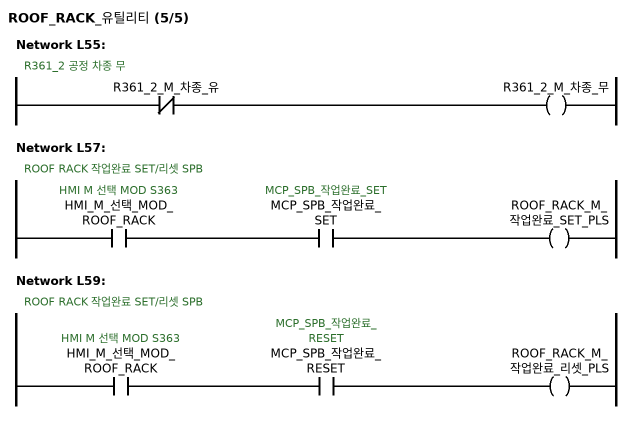
(* [picture p72: ROOF_RACK_유틸리티 rungs L55-L59] *)
(* R361_2 공정 차종 무 *)
(* Rung L55 *)
R361_2_M_차종_무 := NOT R361_2_M_차종_유;
(* ROOF RACK 작업완료 SET/리셋 SPB *)
(* Rung L57 *)
ROOF_RACK_M_작업완료_SET_PLS := HMI_M_선택_MOD_ROOF_RACK AND MCP_SPB_작업완료_SET;
(* ROOF RACK 작업완료 SET/리셋 SPB *)
(* Rung L59 *)
ROOF_RACK_M_작업완료_리셋_PLS := HMI_M_선택_MOD_ROOF_RACK AND MCP_SPB_작업완료_RESET;
END_PROGRAM

PROGRAM ROOF_RACK_차종입력_차종삭제 (* task: 스캔 프로그램 *)
VAR
    INST : TON;
    INST1 : TON;
    INST2 : TON;
    INST3 : TON;
    INST4 : TON;
    INST5 : TON;
END_VAR
VAR_EXTERNAL
    R361_1_I_RB_PLT_최종UNLOAD_완료 : BOOL; (* AT %MW84013.12 *) (* R361_1_I_RB_PLT_최종UNLOAD_완료 *)
    R361_2_I_RB_PLT_최종UNLOAD_완료 : BOOL; (* AT %MW84023.12 *) (* R361_2_I_RB_PLT_최종UNLOAD_완료 *)
END_VAR
VAR_EXTERNAL RETAIN
    R361_1_M_RACK3_프로그램_OK : BOOL; (* AT %MW1563.2 *)
    R361_1_M_RACK4_프로그램_OK : BOOL; (* AT %MW1563.3 *)
    R361_1_M_RACK5_프로그램_OK : BOOL; (* AT %MW1563.4 *)
    R361_1_M_RACK6_프로그램_OK : BOOL; (* AT %MW1563.5 *)
    R361_2_M_RACK1_프로그램_OK : BOOL; (* AT %MW1563.0 *)
    R361_2_M_RACK2_프로그램_OK : BOOL; (* AT %MW1563.1 *)
    ROOF_RACK1_M_HMI입력_차종 : WORD; (* AT %MW501 *)
    ROOF_RACK1_M_랙감지_유 : BOOL; (* AT %MW1501.0 *)
    ROOF_RACK1_M_로딩완료 : BOOL; (* AT %MW1561.0 *)
    ROOF_RACK1_M_막장감지_유 : BOOL; (* AT %MW1503.0 *)
    ROOF_RACK1_M_제품수량 : WORD; (* AT %MW511 *)
    ROOF_RACK1_M_차종 : WORD; (* AT %MW1541 *)
    ROOF_RACK2_M_HMI입력_차종 : WORD; (* AT %MW502 *)
    ROOF_RACK2_M_랙감지_유 : BOOL; (* AT %MW1501.2 *)
    ROOF_RACK2_M_로딩완료 : BOOL; (* AT %MW1561.1 *)
    ROOF_RACK2_M_막장감지_유 : BOOL; (* AT %MW1503.2 *)
    ROOF_RACK2_M_제품수량 : WORD; (* AT %MW512 *)
    ROOF_RACK2_M_차종 : WORD; (* AT %MW1542 *)
    ROOF_RACK3_M_HMI입력_차종 : WORD; (* AT %MW503 *)
    ROOF_RACK3_M_랙감지_유 : BOOL; (* AT %MW1501.4 *)
    ROOF_RACK3_M_로딩완료 : BOOL; (* AT %MW1561.2 *)
    ROOF_RACK3_M_막장감지_유 : BOOL; (* AT %MW1503.4 *)
    ROOF_RACK3_M_제품수량 : WORD; (* AT %MW513 *)
    ROOF_RACK3_M_차종 : WORD; (* AT %MW1543 *)
    ROOF_RACK4_M_HMI입력_차종 : WORD; (* AT %MW504 *)
    ROOF_RACK4_M_랙감지_유 : BOOL; (* AT %MW1501.6 *)
    ROOF_RACK4_M_로딩완료 : BOOL; (* AT %MW1561.3 *)
    ROOF_RACK4_M_막장감지_유 : BOOL; (* AT %MW1503.6 *)
    ROOF_RACK4_M_제품수량 : WORD; (* AT %MW514 *)
    ROOF_RACK4_M_차종 : WORD; (* AT %MW1544 *)
    ROOF_RACK5_M_HMI입력_차종 : WORD; (* AT %MW505 *)
    ROOF_RACK5_M_랙감지_유 : BOOL; (* AT %MW1501.8 *)
    ROOF_RACK5_M_로딩완료 : BOOL; (* AT %MW1561.4 *)
    ROOF_RACK5_M_막장감지_유 : BOOL; (* AT %MW1503.8 *)
    ROOF_RACK5_M_제품수량 : WORD; (* AT %MW515 *)
    ROOF_RACK5_M_차종 : WORD; (* AT %MW1545 *)
    ROOF_RACK6_M_HMI입력_차종 : WORD; (* AT %MW506 *)
    ROOF_RACK6_M_랙감지_유 : BOOL; (* AT %MW1501.10 *)
    ROOF_RACK6_M_로딩완료 : BOOL; (* AT %MW1561.5 *)
    ROOF_RACK6_M_막장감지_유 : BOOL; (* AT %MW1503.10 *)
    ROOF_RACK6_M_제품수량 : WORD; (* AT %MW516 *)
    ROOF_RACK6_M_차종 : WORD; (* AT %MW1546 *)
END_VAR
VAR
    _p1 : BOOL;
    _p2 : BOOL;
    _p3 : BOOL;
    _p4 : BOOL;
    _p5 : BOOL;
    _p6 : BOOL;
END_VAR
(* ================================================================= *)
(* ROOF RACK 차종 입력 *)
(* ================================================================= *)
(* ROOF RACK1 차종입력 *)
(* Rung L4: network not rendered *)
(* not connected or not rendered: ROOF_RACK1_M_로딩완료, ROOF_RACK1_M_랙감지_유, ROOF_RACK1_M_막장감지_유, ROOF_RACK1_M_HMI입력_차종, ROOF_RACK1_M_차종, 10, ROOF_RACK1_M_제품수량 *)
(* ROOF RACK2 차종입력 *)
(* Rung L8: network not rendered *)
(* not connected or not rendered: ROOF_RACK2_M_로딩완료, ROOF_RACK2_M_랙감지_유, ROOF_RACK2_M_막장감지_유, ROOF_RACK2_M_HMI입력_차종, ROOF_RACK2_M_차종, 10, ROOF_RACK2_M_제품수량 *)
(* ROOF RACK3 차종입력 *)
(* Rung L12: network not rendered *)
(* not connected or not rendered: ROOF_RACK3_M_로딩완료, ROOF_RACK3_M_랙감지_유, ROOF_RACK3_M_막장감지_유, ROOF_RACK3_M_HMI입력_차종, ROOF_RACK3_M_차종, 10, ROOF_RACK3_M_제품수량 *)
(* ROOF RACK4 차종입력 *)
(* Rung L16: network not rendered *)
(* not connected or not rendered: ROOF_RACK4_M_로딩완료, ROOF_RACK4_M_랙감지_유, ROOF_RACK4_M_막장감지_유, ROOF_RACK4_M_HMI입력_차종, ROOF_RACK4_M_차종, 10, ROOF_RACK4_M_제품수량 *)
(* ROOF RACK5 차종입력 *)
(* Rung L20: network not rendered *)
(* not connected or not rendered: ROOF_RACK5_M_로딩완료, ROOF_RACK5_M_랙감지_유, ROOF_RACK5_M_막장감지_유, ROOF_RACK5_M_HMI입력_차종, ROOF_RACK5_M_차종, 10, ROOF_RACK5_M_제품수량 *)
(* ROOF RACK6 차종입력 *)
(* Rung L24: network not rendered *)
(* not connected or not rendered: ROOF_RACK6_M_로딩완료, ROOF_RACK6_M_랙감지_유, ROOF_RACK6_M_막장감지_유, ROOF_RACK6_M_HMI입력_차종, ROOF_RACK6_M_차종, 10, ROOF_RACK6_M_제품수량 *)

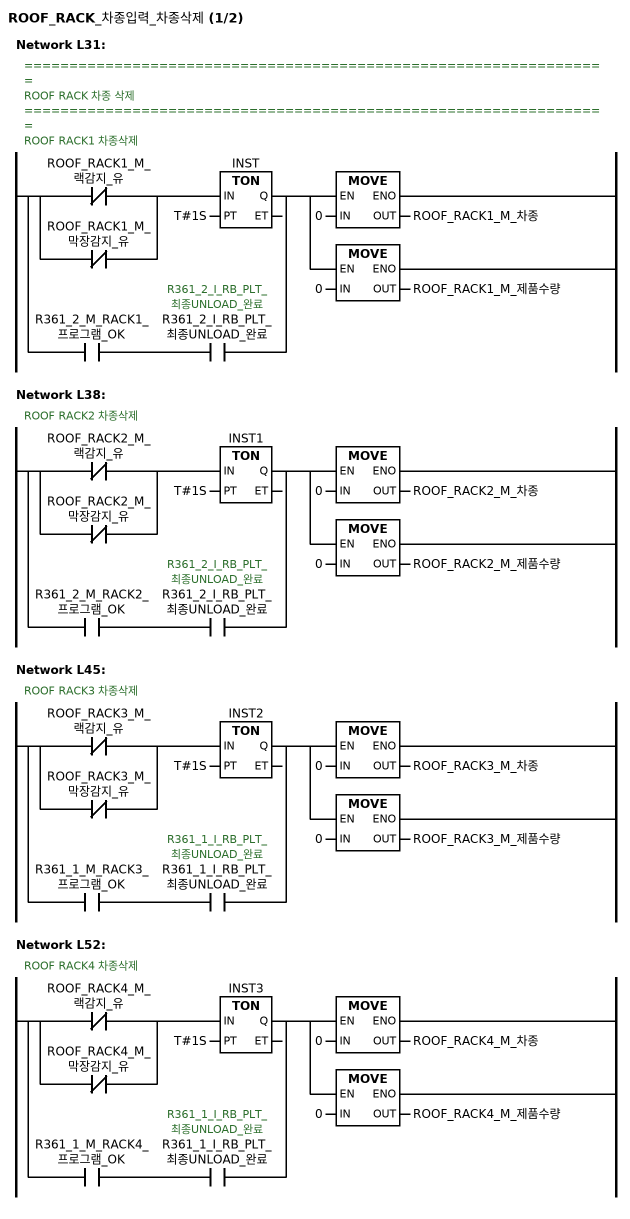
(* ================================================================= *)
(* ROOF RACK 차종 삭제 *)
(* ================================================================= *)
(* ROOF RACK1 차종삭제 *)
(* Rung L31 *)
INST(IN := NOT ROOF_RACK1_M_랙감지_유 OR NOT ROOF_RACK1_M_막장감지_유, PT := T#1S);
_p1 := INST.Q OR (R361_2_M_RACK1_프로그램_OK AND R361_2_I_RB_PLT_최종UNLOAD_완료);
IF _p1 THEN
    ROOF_RACK1_M_차종 := 0;
    ROOF_RACK1_M_제품수량 := 0;
END_IF;
(* ROOF RACK2 차종삭제 *)
(* Rung L38 *)
INST1(IN := NOT ROOF_RACK2_M_랙감지_유 OR NOT ROOF_RACK2_M_막장감지_유, PT := T#1S);
_p2 := INST1.Q OR (R361_2_M_RACK2_프로그램_OK AND R361_2_I_RB_PLT_최종UNLOAD_완료);
IF _p2 THEN
    ROOF_RACK2_M_차종 := 0;
    ROOF_RACK2_M_제품수량 := 0;
END_IF;
(* ROOF RACK3 차종삭제 *)
(* Rung L45 *)
INST2(IN := NOT ROOF_RACK3_M_랙감지_유 OR NOT ROOF_RACK3_M_막장감지_유, PT := T#1S);
_p3 := INST2.Q OR (R361_1_M_RACK3_프로그램_OK AND R361_1_I_RB_PLT_최종UNLOAD_완료);
IF _p3 THEN
    ROOF_RACK3_M_차종 := 0;
    ROOF_RACK3_M_제품수량 := 0;
END_IF;
(* ROOF RACK4 차종삭제 *)
(* Rung L52 *)
INST3(IN := NOT ROOF_RACK4_M_랙감지_유 OR NOT ROOF_RACK4_M_막장감지_유, PT := T#1S);
_p4 := INST3.Q OR (R361_1_M_RACK4_프로그램_OK AND R361_1_I_RB_PLT_최종UNLOAD_완료);
IF _p4 THEN
    ROOF_RACK4_M_차종 := 0;
    ROOF_RACK4_M_제품수량 := 0;
END_IF;

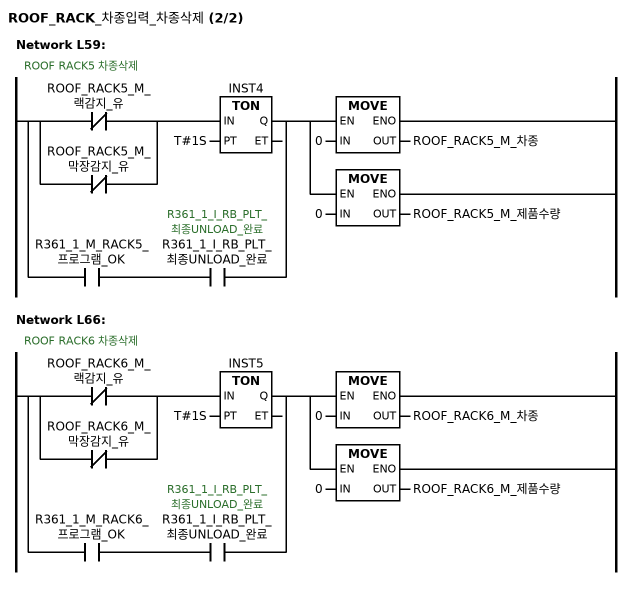
(* ROOF RACK5 차종삭제 *)
(* Rung L59 *)
INST4(IN := NOT ROOF_RACK5_M_랙감지_유 OR NOT ROOF_RACK5_M_막장감지_유, PT := T#1S);
_p5 := INST4.Q OR (R361_1_M_RACK5_프로그램_OK AND R361_1_I_RB_PLT_최종UNLOAD_완료);
IF _p5 THEN
    ROOF_RACK5_M_차종 := 0;
    ROOF_RACK5_M_제품수량 := 0;
END_IF;
(* ROOF RACK6 차종삭제 *)
(* Rung L66 *)
INST5(IN := NOT ROOF_RACK6_M_랙감지_유 OR NOT ROOF_RACK6_M_막장감지_유, PT := T#1S);
_p6 := INST5.Q OR (R361_1_M_RACK6_프로그램_OK AND R361_1_I_RB_PLT_최종UNLOAD_완료);
IF _p6 THEN
    ROOF_RACK6_M_차종 := 0;
    ROOF_RACK6_M_제품수량 := 0;
END_IF;
END_PROGRAM

PROGRAM ROOF_RACK_유_무 (* task: 스캔 프로그램 *)
VAR
    INST : TON;
    INST1 : TON;
    INST2 : TON;
    INST3 : TON;
    INST4 : TON;
    INST5 : TON;
    INST6 : TON;
END_VAR
VAR_EXTERNAL RETAIN
    ROOF_RACK1_M_랙감지_무 : BOOL; (* AT %MW1501.1 *)
    ROOF_RACK1_M_랙감지_유 : BOOL; (* AT %MW1501.0 *)
    ROOF_RACK1_M_로딩완료 : BOOL; (* AT %MW1561.0 *)
    ROOF_RACK1_M_막장감지_무 : BOOL; (* AT %MW1503.1 *)
    ROOF_RACK1_M_막장감지_유 : BOOL; (* AT %MW1503.0 *)
    ROOF_RACK1_M_차종 : WORD; (* AT %MW1541 *)
    ROOF_RACK1_M_차종_무 : BOOL; (* AT %MW1540.1 *)
    ROOF_RACK1_M_차종_유 : BOOL; (* AT %MW1540.0 *)
    ROOF_RACK2_M_랙감지_무 : BOOL; (* AT %MW1501.3 *)
    ROOF_RACK2_M_랙감지_유 : BOOL; (* AT %MW1501.2 *)
    ROOF_RACK2_M_로딩완료 : BOOL; (* AT %MW1561.1 *)
    ROOF_RACK2_M_막장감지_무 : BOOL; (* AT %MW1503.3 *)
    ROOF_RACK2_M_막장감지_유 : BOOL; (* AT %MW1503.2 *)
    ROOF_RACK2_M_차종 : WORD; (* AT %MW1542 *)
    ROOF_RACK2_M_차종_무 : BOOL; (* AT %MW1540.3 *)
    ROOF_RACK2_M_차종_유 : BOOL; (* AT %MW1540.2 *)
    ROOF_RACK3_M_랙감지_무 : BOOL; (* AT %MW1501.5 *)
    ROOF_RACK3_M_랙감지_유 : BOOL; (* AT %MW1501.4 *)
    ROOF_RACK3_M_로딩완료 : BOOL; (* AT %MW1561.2 *)
    ROOF_RACK3_M_막장감지_무 : BOOL; (* AT %MW1503.5 *)
    ROOF_RACK3_M_막장감지_유 : BOOL; (* AT %MW1503.4 *)
    ROOF_RACK3_M_차종 : WORD; (* AT %MW1543 *)
    ROOF_RACK3_M_차종_무 : BOOL; (* AT %MW1540.5 *)
    ROOF_RACK3_M_차종_유 : BOOL; (* AT %MW1540.4 *)
    ROOF_RACK4_M_랙감지_무 : BOOL; (* AT %MW1501.7 *)
    ROOF_RACK4_M_랙감지_유 : BOOL; (* AT %MW1501.6 *)
    ROOF_RACK4_M_로딩완료 : BOOL; (* AT %MW1561.3 *)
    ROOF_RACK4_M_막장감지_무 : BOOL; (* AT %MW1503.7 *)
    ROOF_RACK4_M_막장감지_유 : BOOL; (* AT %MW1503.6 *)
    ROOF_RACK4_M_차종 : WORD; (* AT %MW1544 *)
    ROOF_RACK4_M_차종_무 : BOOL; (* AT %MW1540.7 *)
    ROOF_RACK4_M_차종_유 : BOOL; (* AT %MW1540.6 *)
    ROOF_RACK5_M_랙감지_무 : BOOL; (* AT %MW1501.9 *)
    ROOF_RACK5_M_랙감지_유 : BOOL; (* AT %MW1501.8 *)
    ROOF_RACK5_M_로딩완료 : BOOL; (* AT %MW1561.4 *)
    ROOF_RACK5_M_막장감지_무 : BOOL; (* AT %MW1503.9 *)
    ROOF_RACK5_M_막장감지_유 : BOOL; (* AT %MW1503.8 *)
    ROOF_RACK5_M_차종 : WORD; (* AT %MW1545 *)
    ROOF_RACK5_M_차종_무 : BOOL; (* AT %MW1540.9 *)
    ROOF_RACK5_M_차종_유 : BOOL; (* AT %MW1540.8 *)
    ROOF_RACK6_M_랙감지_무 : BOOL; (* AT %MW1501.11 *)
    ROOF_RACK6_M_랙감지_유 : BOOL; (* AT %MW1501.10 *)
    ROOF_RACK6_M_로딩완료 : BOOL; (* AT %MW1561.5 *)
    ROOF_RACK6_M_막장감지_무 : BOOL; (* AT %MW1503.11 *)
    ROOF_RACK6_M_막장감지_유 : BOOL; (* AT %MW1503.10 *)
    ROOF_RACK6_M_차종 : WORD; (* AT %MW1546 *)
    ROOF_RACK6_M_차종_무 : BOOL; (* AT %MW1540.11 *)
    ROOF_RACK6_M_차종_유 : BOOL; (* AT %MW1540.10 *)
END_VAR
VAR_EXTERNAL
    ROOF_RACK1_PRS_랙감지1 : BOOL; (* AT %MW87400.0 *) (* ROOF RACK1 PRS 랙감지1 *)
    ROOF_RACK1_PRS_랙감지2 : BOOL; (* AT %MW87400.1 *) (* ROOF RACK1 PRS 랙감지2 *)
    ROOF_RACK1_PRS_막장감지 : BOOL; (* AT %MW87400.2 *) (* ROOF RACK1 PRS 막장감지 *)
    ROOF_RACK2_PRS_랙감지1 : BOOL; (* AT %MW87400.8 *) (* ROOF RACK2 PRS 랙감지1 *)
    ROOF_RACK2_PRS_랙감지2 : BOOL; (* AT %MW87400.9 *) (* ROOF RACK2 PRS 랙감지2 *)
    ROOF_RACK2_PRS_막장감지 : BOOL; (* AT %MW87400.10 *) (* ROOF RACK2 PRS 막장감지 *)
    ROOF_RACK3_PRS_랙감지1 : BOOL; (* AT %MW87401.0 *) (* ROOF RACK3 PRS 랙감지1 *)
    ROOF_RACK3_PRS_랙감지2 : BOOL; (* AT %MW87401.1 *) (* ROOF RACK3 PRS 랙감지2 *)
    ROOF_RACK3_PRS_막장감지 : BOOL; (* AT %MW87401.2 *) (* ROOF RACK3 PRS 막장감지 *)
    ROOF_RACK4_PRS_랙감지1 : BOOL; (* AT %MW87450.0 *) (* ROOF RACK4 PRS 랙감지1 *)
    ROOF_RACK4_PRS_랙감지2 : BOOL; (* AT %MW87450.1 *) (* ROOF RACK4 PRS 랙감지2 *)
    ROOF_RACK4_PRS_막장감지 : BOOL; (* AT %MW87450.2 *) (* ROOF RACK4 PRS 막장감지 *)
    ROOF_RACK5_PRS_랙감지1 : BOOL; (* AT %MW87450.8 *) (* ROOF RACK5 PRS 랙감지1 *)
    ROOF_RACK5_PRS_랙감지2 : BOOL; (* AT %MW87450.9 *) (* ROOF RACK5 PRS 랙감지2 *)
    ROOF_RACK5_PRS_막장감지 : BOOL; (* AT %MW87450.10 *) (* ROOF RACK5 PRS 막장감지 *)
    ROOF_RACK6_PRS_랙감지1 : BOOL; (* AT %MW87451.0 *) (* ROOF RACK6 PRS 랙감지1 *)
    ROOF_RACK6_PRS_랙감지2 : BOOL; (* AT %MW87451.1 *) (* ROOF RACK6 PRS 랙감지2 *)
    ROOF_RACK6_PRS_막장감지 : BOOL; (* AT %MW87451.2 *) (* ROOF RACK6 PRS 막장감지 *)
END_VAR

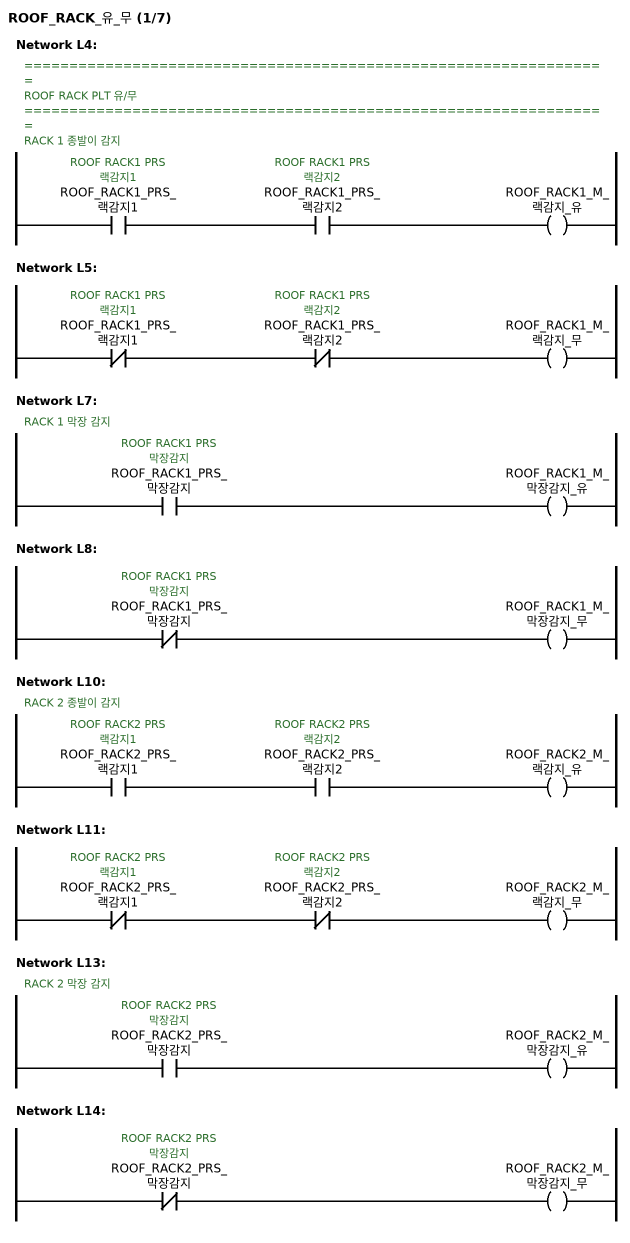
(* ================================================================= *)
(* ROOF RACK PLT 유/무 *)
(* ================================================================= *)
(* RACK 1 종발이 감지 *)
(* Rung L4 *)
ROOF_RACK1_M_랙감지_유 := ROOF_RACK1_PRS_랙감지1 AND ROOF_RACK1_PRS_랙감지2;
(* Rung L5 *)
ROOF_RACK1_M_랙감지_무 := NOT ROOF_RACK1_PRS_랙감지1 AND NOT ROOF_RACK1_PRS_랙감지2;
(* RACK 1 막장 감지 *)
(* Rung L7 *)
ROOF_RACK1_M_막장감지_유 := ROOF_RACK1_PRS_막장감지;
(* Rung L8 *)
ROOF_RACK1_M_막장감지_무 := NOT ROOF_RACK1_PRS_막장감지;
(* RACK 2 종발이 감지 *)
(* Rung L10 *)
ROOF_RACK2_M_랙감지_유 := ROOF_RACK2_PRS_랙감지1 AND ROOF_RACK2_PRS_랙감지2;
(* Rung L11 *)
ROOF_RACK2_M_랙감지_무 := NOT ROOF_RACK2_PRS_랙감지1 AND NOT ROOF_RACK2_PRS_랙감지2;
(* RACK 2 막장 감지 *)
(* Rung L13 *)
ROOF_RACK2_M_막장감지_유 := ROOF_RACK2_PRS_막장감지;
(* Rung L14 *)
ROOF_RACK2_M_막장감지_무 := NOT ROOF_RACK2_PRS_막장감지;

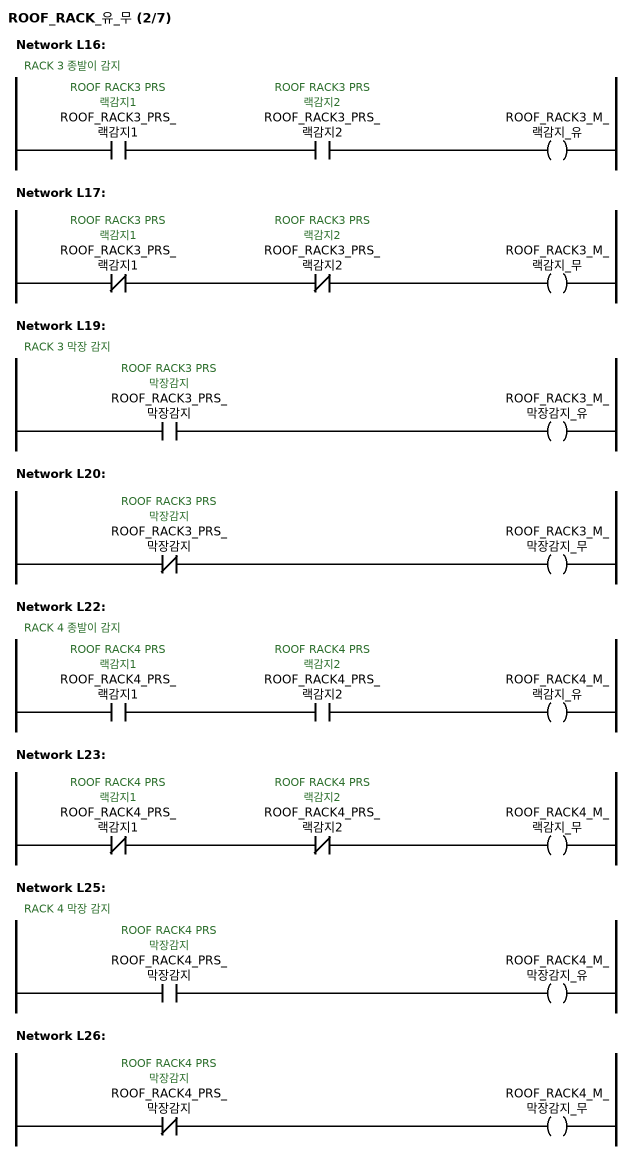
(* RACK 3 종발이 감지 *)
(* Rung L16 *)
ROOF_RACK3_M_랙감지_유 := ROOF_RACK3_PRS_랙감지1 AND ROOF_RACK3_PRS_랙감지2;
(* Rung L17 *)
ROOF_RACK3_M_랙감지_무 := NOT ROOF_RACK3_PRS_랙감지1 AND NOT ROOF_RACK3_PRS_랙감지2;
(* RACK 3 막장 감지 *)
(* Rung L19 *)
ROOF_RACK3_M_막장감지_유 := ROOF_RACK3_PRS_막장감지;
(* Rung L20 *)
ROOF_RACK3_M_막장감지_무 := NOT ROOF_RACK3_PRS_막장감지;
(* RACK 4 종발이 감지 *)
(* Rung L22 *)
ROOF_RACK4_M_랙감지_유 := ROOF_RACK4_PRS_랙감지1 AND ROOF_RACK4_PRS_랙감지2;
(* Rung L23 *)
ROOF_RACK4_M_랙감지_무 := NOT ROOF_RACK4_PRS_랙감지1 AND NOT ROOF_RACK4_PRS_랙감지2;
(* RACK 4 막장 감지 *)
(* Rung L25 *)
ROOF_RACK4_M_막장감지_유 := ROOF_RACK4_PRS_막장감지;
(* Rung L26 *)
ROOF_RACK4_M_막장감지_무 := NOT ROOF_RACK4_PRS_막장감지;

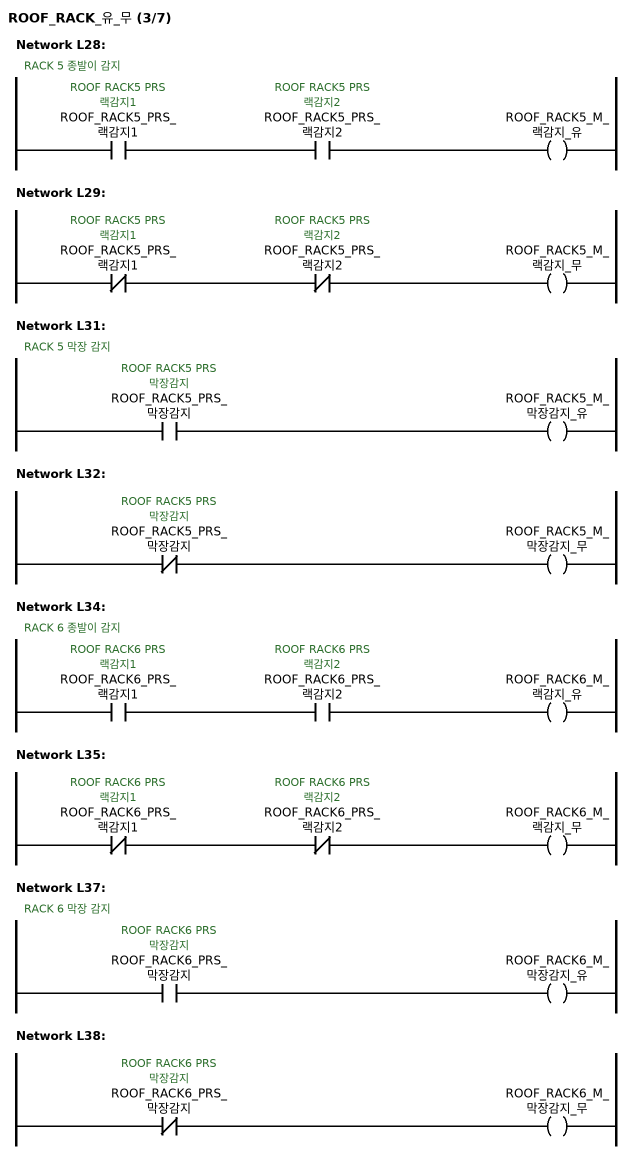
(* RACK 5 종발이 감지 *)
(* Rung L28 *)
ROOF_RACK5_M_랙감지_유 := ROOF_RACK5_PRS_랙감지1 AND ROOF_RACK5_PRS_랙감지2;
(* Rung L29 *)
ROOF_RACK5_M_랙감지_무 := NOT ROOF_RACK5_PRS_랙감지1 AND NOT ROOF_RACK5_PRS_랙감지2;
(* RACK 5 막장 감지 *)
(* Rung L31 *)
ROOF_RACK5_M_막장감지_유 := ROOF_RACK5_PRS_막장감지;
(* Rung L32 *)
ROOF_RACK5_M_막장감지_무 := NOT ROOF_RACK5_PRS_막장감지;
(* RACK 6 종발이 감지 *)
(* Rung L34 *)
ROOF_RACK6_M_랙감지_유 := ROOF_RACK6_PRS_랙감지1 AND ROOF_RACK6_PRS_랙감지2;
(* Rung L35 *)
ROOF_RACK6_M_랙감지_무 := NOT ROOF_RACK6_PRS_랙감지1 AND NOT ROOF_RACK6_PRS_랙감지2;
(* RACK 6 막장 감지 *)
(* Rung L37 *)
ROOF_RACK6_M_막장감지_유 := ROOF_RACK6_PRS_막장감지;
(* Rung L38 *)
ROOF_RACK6_M_막장감지_무 := NOT ROOF_RACK6_PRS_막장감지;

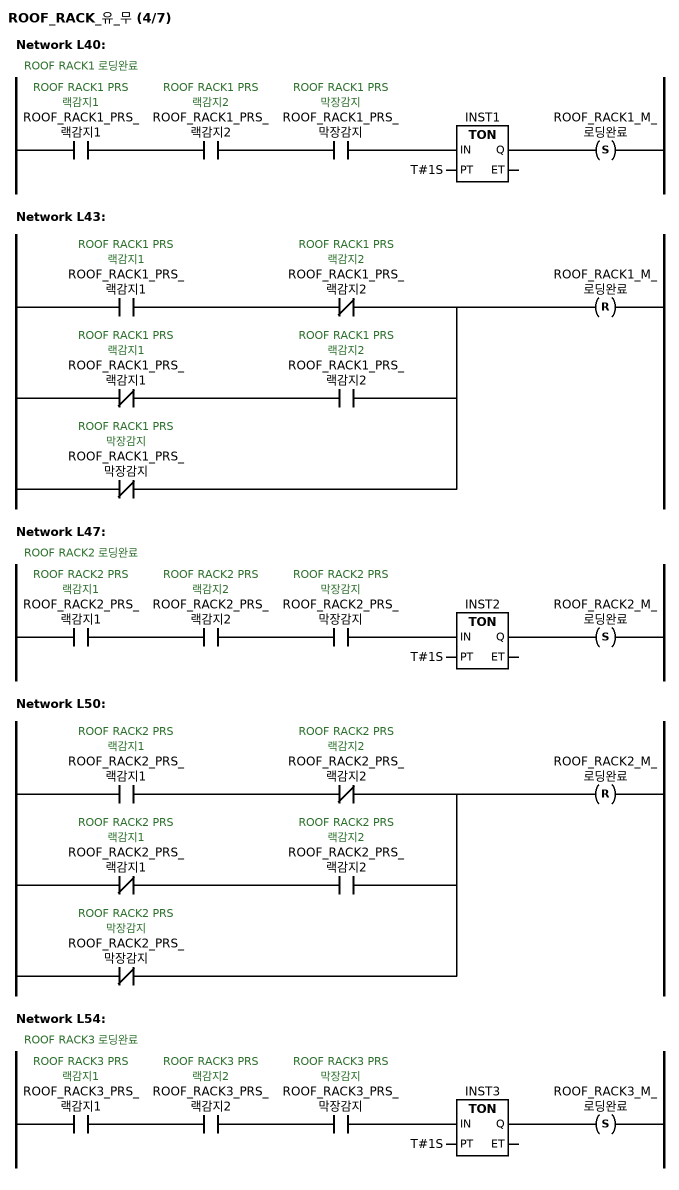
(* ROOF RACK1 로딩완료 *)
(* Rung L40 *)
INST1(IN := ROOF_RACK1_PRS_랙감지1 AND ROOF_RACK1_PRS_랙감지2 AND ROOF_RACK1_PRS_막장감지, PT := T#1S);
IF INST1.Q THEN ROOF_RACK1_M_로딩완료 := TRUE; END_IF;
(* Rung L43 *)
IF (ROOF_RACK1_PRS_랙감지1 AND NOT ROOF_RACK1_PRS_랙감지2) OR (NOT ROOF_RACK1_PRS_랙감지1 AND ROOF_RACK1_PRS_랙감지2) OR NOT ROOF_RACK1_PRS_막장감지 THEN
    ROOF_RACK1_M_로딩완료 := FALSE;
END_IF;
(* ROOF RACK2 로딩완료 *)
(* Rung L47 *)
INST2(IN := ROOF_RACK2_PRS_랙감지1 AND ROOF_RACK2_PRS_랙감지2 AND ROOF_RACK2_PRS_막장감지, PT := T#1S);
IF INST2.Q THEN ROOF_RACK2_M_로딩완료 := TRUE; END_IF;
(* Rung L50 *)
IF (ROOF_RACK2_PRS_랙감지1 AND NOT ROOF_RACK2_PRS_랙감지2) OR (NOT ROOF_RACK2_PRS_랙감지1 AND ROOF_RACK2_PRS_랙감지2) OR NOT ROOF_RACK2_PRS_막장감지 THEN
    ROOF_RACK2_M_로딩완료 := FALSE;
END_IF;
(* ROOF RACK3 로딩완료 *)
(* Rung L54 *)
INST3(IN := ROOF_RACK3_PRS_랙감지1 AND ROOF_RACK3_PRS_랙감지2 AND ROOF_RACK3_PRS_막장감지, PT := T#1S);
IF INST3.Q THEN ROOF_RACK3_M_로딩완료 := TRUE; END_IF;

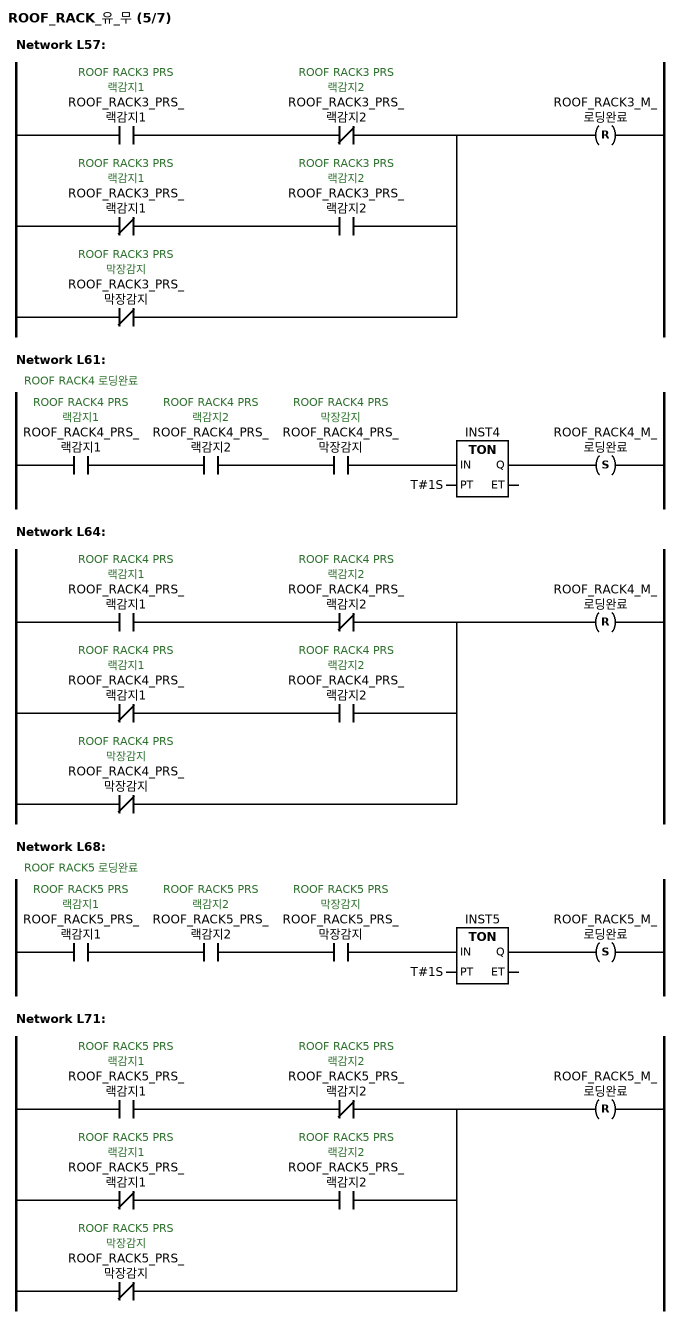
(* Rung L57 *)
IF (ROOF_RACK3_PRS_랙감지1 AND NOT ROOF_RACK3_PRS_랙감지2) OR (NOT ROOF_RACK3_PRS_랙감지1 AND ROOF_RACK3_PRS_랙감지2) OR NOT ROOF_RACK3_PRS_막장감지 THEN
    ROOF_RACK3_M_로딩완료 := FALSE;
END_IF;
(* ROOF RACK4 로딩완료 *)
(* Rung L61 *)
INST4(IN := ROOF_RACK4_PRS_랙감지1 AND ROOF_RACK4_PRS_랙감지2 AND ROOF_RACK4_PRS_막장감지, PT := T#1S);
IF INST4.Q THEN ROOF_RACK4_M_로딩완료 := TRUE; END_IF;
(* Rung L64 *)
IF (ROOF_RACK4_PRS_랙감지1 AND NOT ROOF_RACK4_PRS_랙감지2) OR (NOT ROOF_RACK4_PRS_랙감지1 AND ROOF_RACK4_PRS_랙감지2) OR NOT ROOF_RACK4_PRS_막장감지 THEN
    ROOF_RACK4_M_로딩완료 := FALSE;
END_IF;
(* ROOF RACK5 로딩완료 *)
(* Rung L68 *)
INST5(IN := ROOF_RACK5_PRS_랙감지1 AND ROOF_RACK5_PRS_랙감지2 AND ROOF_RACK5_PRS_막장감지, PT := T#1S);
IF INST5.Q THEN ROOF_RACK5_M_로딩완료 := TRUE; END_IF;
(* Rung L71 *)
IF (ROOF_RACK5_PRS_랙감지1 AND NOT ROOF_RACK5_PRS_랙감지2) OR (NOT ROOF_RACK5_PRS_랙감지1 AND ROOF_RACK5_PRS_랙감지2) OR NOT ROOF_RACK5_PRS_막장감지 THEN
    ROOF_RACK5_M_로딩완료 := FALSE;
END_IF;

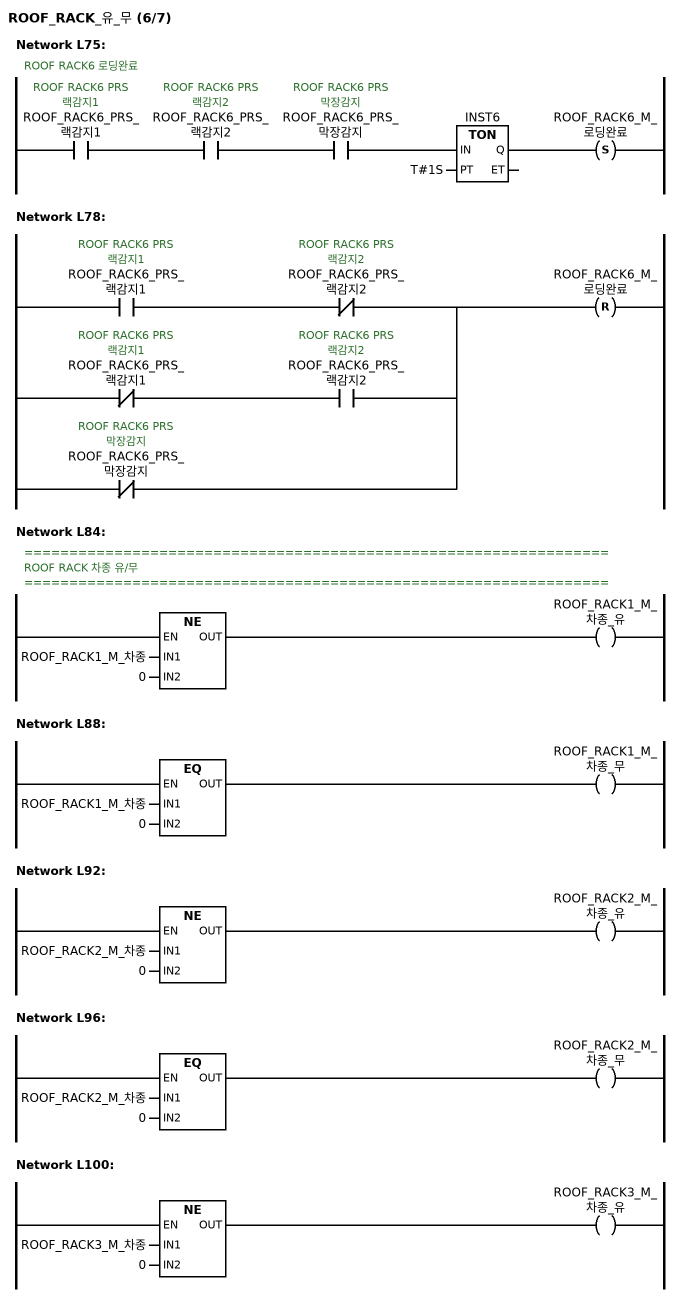
(* ROOF RACK6 로딩완료 *)
(* Rung L75 *)
INST6(IN := ROOF_RACK6_PRS_랙감지1 AND ROOF_RACK6_PRS_랙감지2 AND ROOF_RACK6_PRS_막장감지, PT := T#1S);
IF INST6.Q THEN ROOF_RACK6_M_로딩완료 := TRUE; END_IF;
(* Rung L78 *)
IF (ROOF_RACK6_PRS_랙감지1 AND NOT ROOF_RACK6_PRS_랙감지2) OR (NOT ROOF_RACK6_PRS_랙감지1 AND ROOF_RACK6_PRS_랙감지2) OR NOT ROOF_RACK6_PRS_막장감지 THEN
    ROOF_RACK6_M_로딩완료 := FALSE;
END_IF;
(* ================================================================= *)
(* ROOF RACK 차종 유/무 *)
(* ================================================================= *)
(* Rung L84 *)
ROOF_RACK1_M_차종_유 := ROOF_RACK1_M_차종 <> 0;
(* Rung L88 *)
ROOF_RACK1_M_차종_무 := ROOF_RACK1_M_차종 = 0;
(* Rung L92 *)
ROOF_RACK2_M_차종_유 := ROOF_RACK2_M_차종 <> 0;
(* Rung L96 *)
ROOF_RACK2_M_차종_무 := ROOF_RACK2_M_차종 = 0;
(* Rung L100 *)
ROOF_RACK3_M_차종_유 := ROOF_RACK3_M_차종 <> 0;

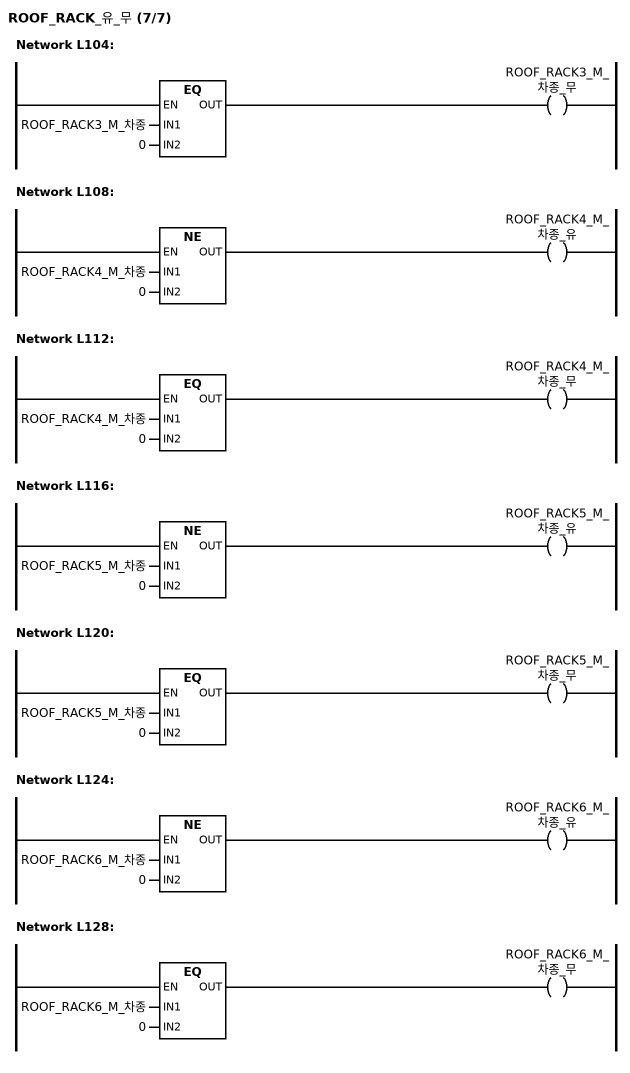
(* Rung L104 *)
ROOF_RACK3_M_차종_무 := ROOF_RACK3_M_차종 = 0;
(* Rung L108 *)
ROOF_RACK4_M_차종_유 := ROOF_RACK4_M_차종 <> 0;
(* Rung L112 *)
ROOF_RACK4_M_차종_무 := ROOF_RACK4_M_차종 = 0;
(* Rung L116 *)
ROOF_RACK5_M_차종_유 := ROOF_RACK5_M_차종 <> 0;
(* Rung L120 *)
ROOF_RACK5_M_차종_무 := ROOF_RACK5_M_차종 = 0;
(* Rung L124 *)
ROOF_RACK6_M_차종_유 := ROOF_RACK6_M_차종 <> 0;
(* Rung L128 *)
ROOF_RACK6_M_차종_무 := ROOF_RACK6_M_차종 = 0;
END_PROGRAM

PROGRAM ROOF_RACK_우선순위 (* task: 스캔 프로그램 *)
VAR_EXTERNAL RETAIN
    ROOF_RACK1_M_랙감지_유 : BOOL; (* AT %MW1501.0 *)
    ROOF_RACK1_M_로딩완료 : BOOL; (* AT %MW1561.0 *)
    ROOF_RACK1_M_막장감지_유 : BOOL; (* AT %MW1503.0 *)
    ROOF_RACK1_M_차종_유 : BOOL; (* AT %MW1540.0 *)
    ROOF_RACK2_M_랙감지_유 : BOOL; (* AT %MW1501.2 *)
    ROOF_RACK2_M_로딩완료 : BOOL; (* AT %MW1561.1 *)
    ROOF_RACK2_M_막장감지_유 : BOOL; (* AT %MW1503.2 *)
    ROOF_RACK2_M_차종_유 : BOOL; (* AT %MW1540.2 *)
    ROOF_RACK3_M_랙감지_유 : BOOL; (* AT %MW1501.4 *)
    ROOF_RACK3_M_로딩완료 : BOOL; (* AT %MW1561.2 *)
    ROOF_RACK3_M_막장감지_유 : BOOL; (* AT %MW1503.4 *)
    ROOF_RACK3_M_차종_유 : BOOL; (* AT %MW1540.4 *)
    ROOF_RACK4_M_랙감지_유 : BOOL; (* AT %MW1501.6 *)
    ROOF_RACK4_M_로딩완료 : BOOL; (* AT %MW1561.3 *)
    ROOF_RACK4_M_막장감지_유 : BOOL; (* AT %MW1503.6 *)
    ROOF_RACK4_M_차종_유 : BOOL; (* AT %MW1540.6 *)
    ROOF_RACK5_M_랙감지_유 : BOOL; (* AT %MW1501.8 *)
    ROOF_RACK5_M_로딩완료 : BOOL; (* AT %MW1561.4 *)
    ROOF_RACK5_M_막장감지_유 : BOOL; (* AT %MW1503.8 *)
    ROOF_RACK5_M_차종_유 : BOOL; (* AT %MW1540.8 *)
    ROOF_RACK6_M_랙감지_유 : BOOL; (* AT %MW1501.10 *)
    ROOF_RACK6_M_로딩완료 : BOOL; (* AT %MW1561.5 *)
    ROOF_RACK6_M_막장감지_유 : BOOL; (* AT %MW1503.10 *)
    ROOF_RACK6_M_차종_유 : BOOL; (* AT %MW1540.10 *)
    ROOF_RACK_M_우선순위_버퍼1 : WORD; (* AT %MW1551 *)
    ROOF_RACK_M_우선순위_버퍼2 : WORD; (* AT %MW1552 *)
    ROOF_RACK_M_우선순위_버퍼3 : WORD; (* AT %MW1553 *)
    ROOF_RACK_M_우선순위_버퍼4 : WORD; (* AT %MW1554 *)
    ROOF_RACK_M_우선순위_버퍼5 : WORD; (* AT %MW1555 *)
    ROOF_RACK_M_우선순위_버퍼6 : WORD; (* AT %MW1556 *)
END_VAR
VAR
    _p1 : BOOL;
    _t2 : BOOL;
    _t3 : BOOL;
    _t4 : BOOL;
    _t5 : BOOL;
    _t6 : BOOL;
    _t7 : BOOL;
    _p8 : BOOL;
    _t9 : BOOL;
    _t10 : BOOL;
    _t11 : BOOL;
    _t12 : BOOL;
    _t13 : BOOL;
    _t14 : BOOL;
    _p15 : BOOL;
    _t16 : BOOL;
    _t17 : BOOL;
    _t18 : BOOL;
    _t19 : BOOL;
    _t20 : BOOL;
    _t21 : BOOL;
    _p22 : BOOL;
    _t23 : BOOL;
    _t24 : BOOL;
    _t25 : BOOL;
    _t26 : BOOL;
    _t27 : BOOL;
    _t28 : BOOL;
    _p29 : BOOL;
    _t30 : BOOL;
    _t31 : BOOL;
    _t32 : BOOL;
    _t33 : BOOL;
    _t34 : BOOL;
    _t35 : BOOL;
    _p36 : BOOL;
    _t37 : BOOL;
    _t38 : BOOL;
    _t39 : BOOL;
    _t40 : BOOL;
    _t41 : BOOL;
    _t42 : BOOL;
END_VAR
(* ================================================================= *)
(* ROOF RACK PLT 우선순위 *)
(* ================================================================= *)
(* 랙방번호 우선순위 버퍼6 *)
(* Rung L4: network not rendered *)
(* not connected or not rendered: ROOF_RACK1_M_로딩완료, ROOF_RACK1_M_랙감지_유, ROOF_RACK1_M_막장감지_유, ROOF_RACK1_M_차종_유, ROOF_RACK2_M_로딩완료, ROOF_RACK2_M_랙감지_유, ROOF_RACK2_M_막장감지_유, ROOF_RACK2_M_차종_유, ROOF_RACK3_M_로딩완료, ROOF_RACK3_M_랙감지_유, ROOF_RACK3_M_막장감지_유, ROOF_RACK3_M_차종_유, ROOF_RACK4_M_로딩완료, ROOF_RACK4_M_랙감지_유, ROOF_RACK4_M_막장감지_유, ROOF_RACK4_M_차종_유, ROOF_RACK5_M_로딩완료, ROOF_RACK5_M_랙감지_유, ROOF_RACK5_M_막장감지_유, ROOF_RACK5_M_차종_유, ROOF_RACK6_M_로딩완료, ROOF_RACK6_M_랙감지_유, ROOF_RACK6_M_막장감지_유, ROOF_RACK6_M_차종_유, ROOF_RACK_M_우선순위_버퍼6, 0, 1, ROOF_RACK_M_우선순위_버퍼6, 2, ROOF_RACK_M_우선순위_버퍼6, 3, ROOF_RACK_M_우선순위_버퍼6, ROOF_RACK_M_우선순위_버퍼6, 5, ROOF_RACK_M_우선순위_버퍼6, 6, ROOF_RACK_M_우선순위_버퍼6 *)
(* 랙방번호 우선순위 버퍼6 -> 우선순위버퍼5 *)
(* Rung L24: network not rendered *)
(* not connected or not rendered: ROOF_RACK_M_우선순위_버퍼6, 0, ROOF_RACK_M_우선순위_버퍼5, 0, ROOF_RACK_M_우선순위_버퍼6, ROOF_RACK_M_우선순위_버퍼5, 0, ROOF_RACK_M_우선순위_버퍼6 *)
(* 랙방번호 우선순위 버퍼5 -> 우선순위버퍼4 *)
(* Rung L33: network not rendered *)
(* not connected or not rendered: ROOF_RACK_M_우선순위_버퍼5, 0, ROOF_RACK_M_우선순위_버퍼4, 0, ROOF_RACK_M_우선순위_버퍼5, ROOF_RACK_M_우선순위_버퍼4, 0, ROOF_RACK_M_우선순위_버퍼5 *)
(* 랙방번호 우선순위 버퍼4 -> 우선순위버퍼3 *)
(* Rung L42: network not rendered *)
(* not connected or not rendered: ROOF_RACK_M_우선순위_버퍼4, 0, ROOF_RACK_M_우선순위_버퍼3, 0, ROOF_RACK_M_우선순위_버퍼4, ROOF_RACK_M_우선순위_버퍼3, 0, ROOF_RACK_M_우선순위_버퍼4 *)
(* 랙방번호 우선순위 버퍼3 -> 우선순위버퍼2 *)
(* Rung L51: network not rendered *)
(* not connected or not rendered: ROOF_RACK_M_우선순위_버퍼3, 0, ROOF_RACK_M_우선순위_버퍼2, 0, ROOF_RACK_M_우선순위_버퍼3, ROOF_RACK_M_우선순위_버퍼2, 0, ROOF_RACK_M_우선순위_버퍼3 *)
(* 랙방번호 우선순위 버퍼2 -> 우선순위버퍼1 *)
(* Rung L60: network not rendered *)
(* not connected or not rendered: ROOF_RACK_M_우선순위_버퍼2, ROOF_RACK_M_우선순위_버퍼1, ROOF_RACK_M_우선순위_버퍼2, ROOF_RACK_M_우선순위_버퍼1, ROOF_RACK_M_우선순위_버퍼2 *)

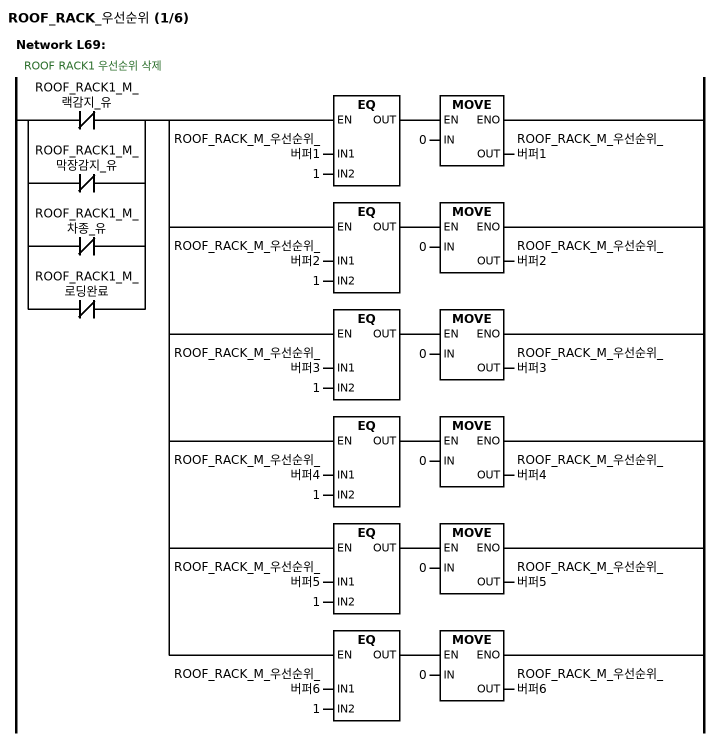
(* ROOF RACK1 우선순위 삭제 *)
(* Rung L69 *)
_p1 := NOT ROOF_RACK1_M_랙감지_유 OR NOT ROOF_RACK1_M_막장감지_유 OR NOT ROOF_RACK1_M_차종_유 OR NOT ROOF_RACK1_M_로딩완료;
IF _p1 THEN _t2 := ROOF_RACK_M_우선순위_버퍼1 = 1; END_IF;
IF _t2 THEN ROOF_RACK_M_우선순위_버퍼1 := 0; END_IF;
IF _p1 THEN _t3 := ROOF_RACK_M_우선순위_버퍼2 = 1; END_IF;
IF _t3 THEN ROOF_RACK_M_우선순위_버퍼2 := 0; END_IF;
IF _p1 THEN _t4 := ROOF_RACK_M_우선순위_버퍼3 = 1; END_IF;
IF _t4 THEN ROOF_RACK_M_우선순위_버퍼3 := 0; END_IF;
IF _p1 THEN _t5 := ROOF_RACK_M_우선순위_버퍼4 = 1; END_IF;
IF _t5 THEN ROOF_RACK_M_우선순위_버퍼4 := 0; END_IF;
IF _p1 THEN _t6 := ROOF_RACK_M_우선순위_버퍼5 = 1; END_IF;
IF _t6 THEN ROOF_RACK_M_우선순위_버퍼5 := 0; END_IF;
IF _p1 THEN _t7 := ROOF_RACK_M_우선순위_버퍼6 = 1; END_IF;
IF _t7 THEN ROOF_RACK_M_우선순위_버퍼6 := 0; END_IF;

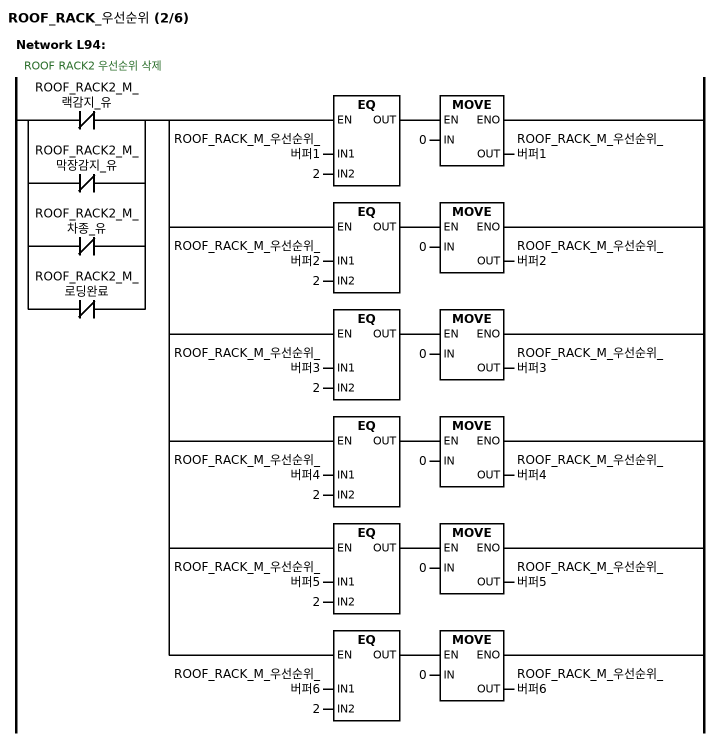
(* ROOF RACK2 우선순위 삭제 *)
(* Rung L94 *)
_p8 := NOT ROOF_RACK2_M_랙감지_유 OR NOT ROOF_RACK2_M_막장감지_유 OR NOT ROOF_RACK2_M_차종_유 OR NOT ROOF_RACK2_M_로딩완료;
IF _p8 THEN _t9 := ROOF_RACK_M_우선순위_버퍼1 = 2; END_IF;
IF _t9 THEN ROOF_RACK_M_우선순위_버퍼1 := 0; END_IF;
IF _p8 THEN _t10 := ROOF_RACK_M_우선순위_버퍼2 = 2; END_IF;
IF _t10 THEN ROOF_RACK_M_우선순위_버퍼2 := 0; END_IF;
IF _p8 THEN _t11 := ROOF_RACK_M_우선순위_버퍼3 = 2; END_IF;
IF _t11 THEN ROOF_RACK_M_우선순위_버퍼3 := 0; END_IF;
IF _p8 THEN _t12 := ROOF_RACK_M_우선순위_버퍼4 = 2; END_IF;
IF _t12 THEN ROOF_RACK_M_우선순위_버퍼4 := 0; END_IF;
IF _p8 THEN _t13 := ROOF_RACK_M_우선순위_버퍼5 = 2; END_IF;
IF _t13 THEN ROOF_RACK_M_우선순위_버퍼5 := 0; END_IF;
IF _p8 THEN _t14 := ROOF_RACK_M_우선순위_버퍼6 = 2; END_IF;
IF _t14 THEN ROOF_RACK_M_우선순위_버퍼6 := 0; END_IF;

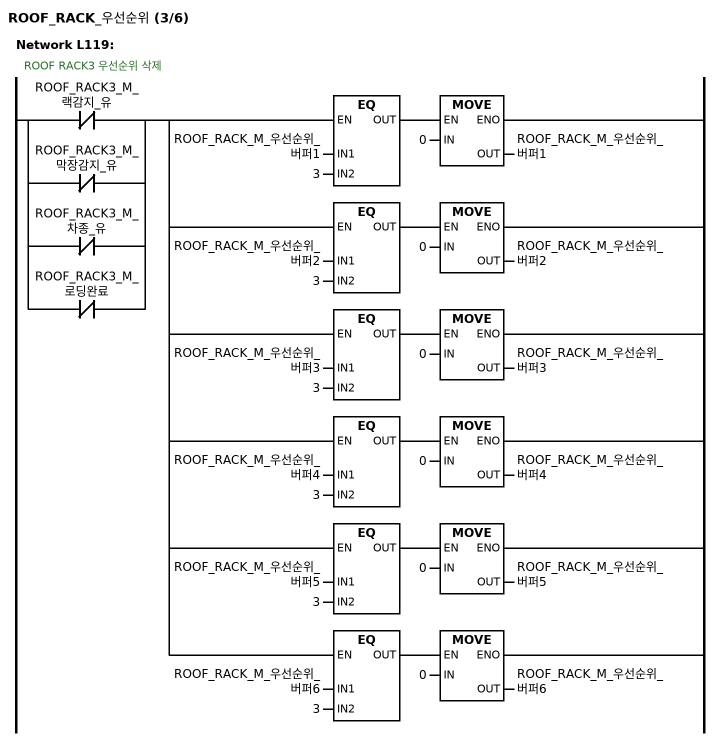
(* ROOF RACK3 우선순위 삭제 *)
(* Rung L119 *)
_p15 := NOT ROOF_RACK3_M_랙감지_유 OR NOT ROOF_RACK3_M_막장감지_유 OR NOT ROOF_RACK3_M_차종_유 OR NOT ROOF_RACK3_M_로딩완료;
IF _p15 THEN _t16 := ROOF_RACK_M_우선순위_버퍼1 = 3; END_IF;
IF _t16 THEN ROOF_RACK_M_우선순위_버퍼1 := 0; END_IF;
IF _p15 THEN _t17 := ROOF_RACK_M_우선순위_버퍼2 = 3; END_IF;
IF _t17 THEN ROOF_RACK_M_우선순위_버퍼2 := 0; END_IF;
IF _p15 THEN _t18 := ROOF_RACK_M_우선순위_버퍼3 = 3; END_IF;
IF _t18 THEN ROOF_RACK_M_우선순위_버퍼3 := 0; END_IF;
IF _p15 THEN _t19 := ROOF_RACK_M_우선순위_버퍼4 = 3; END_IF;
IF _t19 THEN ROOF_RACK_M_우선순위_버퍼4 := 0; END_IF;
IF _p15 THEN _t20 := ROOF_RACK_M_우선순위_버퍼5 = 3; END_IF;
IF _t20 THEN ROOF_RACK_M_우선순위_버퍼5 := 0; END_IF;
IF _p15 THEN _t21 := ROOF_RACK_M_우선순위_버퍼6 = 3; END_IF;
IF _t21 THEN ROOF_RACK_M_우선순위_버퍼6 := 0; END_IF;

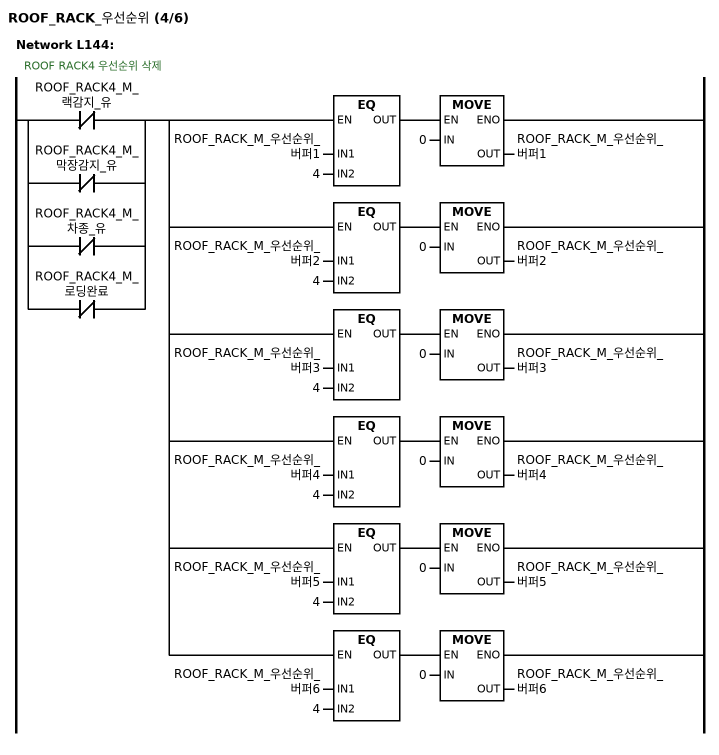
(* ROOF RACK4 우선순위 삭제 *)
(* Rung L144 *)
_p22 := NOT ROOF_RACK4_M_랙감지_유 OR NOT ROOF_RACK4_M_막장감지_유 OR NOT ROOF_RACK4_M_차종_유 OR NOT ROOF_RACK4_M_로딩완료;
IF _p22 THEN _t23 := ROOF_RACK_M_우선순위_버퍼1 = 4; END_IF;
IF _t23 THEN ROOF_RACK_M_우선순위_버퍼1 := 0; END_IF;
IF _p22 THEN _t24 := ROOF_RACK_M_우선순위_버퍼2 = 4; END_IF;
IF _t24 THEN ROOF_RACK_M_우선순위_버퍼2 := 0; END_IF;
IF _p22 THEN _t25 := ROOF_RACK_M_우선순위_버퍼3 = 4; END_IF;
IF _t25 THEN ROOF_RACK_M_우선순위_버퍼3 := 0; END_IF;
IF _p22 THEN _t26 := ROOF_RACK_M_우선순위_버퍼4 = 4; END_IF;
IF _t26 THEN ROOF_RACK_M_우선순위_버퍼4 := 0; END_IF;
IF _p22 THEN _t27 := ROOF_RACK_M_우선순위_버퍼5 = 4; END_IF;
IF _t27 THEN ROOF_RACK_M_우선순위_버퍼5 := 0; END_IF;
IF _p22 THEN _t28 := ROOF_RACK_M_우선순위_버퍼6 = 4; END_IF;
IF _t28 THEN ROOF_RACK_M_우선순위_버퍼6 := 0; END_IF;

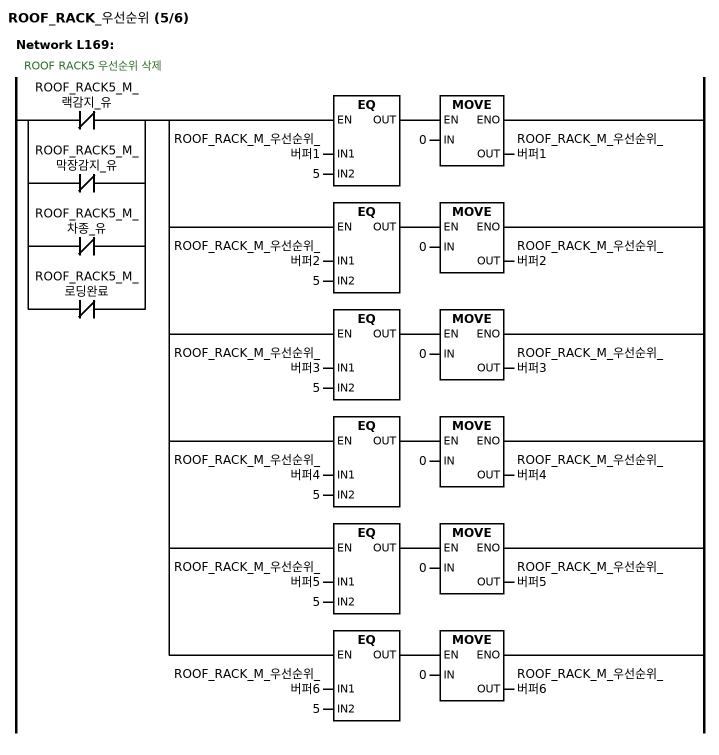
(* ROOF RACK5 우선순위 삭제 *)
(* Rung L169 *)
_p29 := NOT ROOF_RACK5_M_랙감지_유 OR NOT ROOF_RACK5_M_막장감지_유 OR NOT ROOF_RACK5_M_차종_유 OR NOT ROOF_RACK5_M_로딩완료;
IF _p29 THEN _t30 := ROOF_RACK_M_우선순위_버퍼1 = 5; END_IF;
IF _t30 THEN ROOF_RACK_M_우선순위_버퍼1 := 0; END_IF;
IF _p29 THEN _t31 := ROOF_RACK_M_우선순위_버퍼2 = 5; END_IF;
IF _t31 THEN ROOF_RACK_M_우선순위_버퍼2 := 0; END_IF;
IF _p29 THEN _t32 := ROOF_RACK_M_우선순위_버퍼3 = 5; END_IF;
IF _t32 THEN ROOF_RACK_M_우선순위_버퍼3 := 0; END_IF;
IF _p29 THEN _t33 := ROOF_RACK_M_우선순위_버퍼4 = 5; END_IF;
IF _t33 THEN ROOF_RACK_M_우선순위_버퍼4 := 0; END_IF;
IF _p29 THEN _t34 := ROOF_RACK_M_우선순위_버퍼5 = 5; END_IF;
IF _t34 THEN ROOF_RACK_M_우선순위_버퍼5 := 0; END_IF;
IF _p29 THEN _t35 := ROOF_RACK_M_우선순위_버퍼6 = 5; END_IF;
IF _t35 THEN ROOF_RACK_M_우선순위_버퍼6 := 0; END_IF;

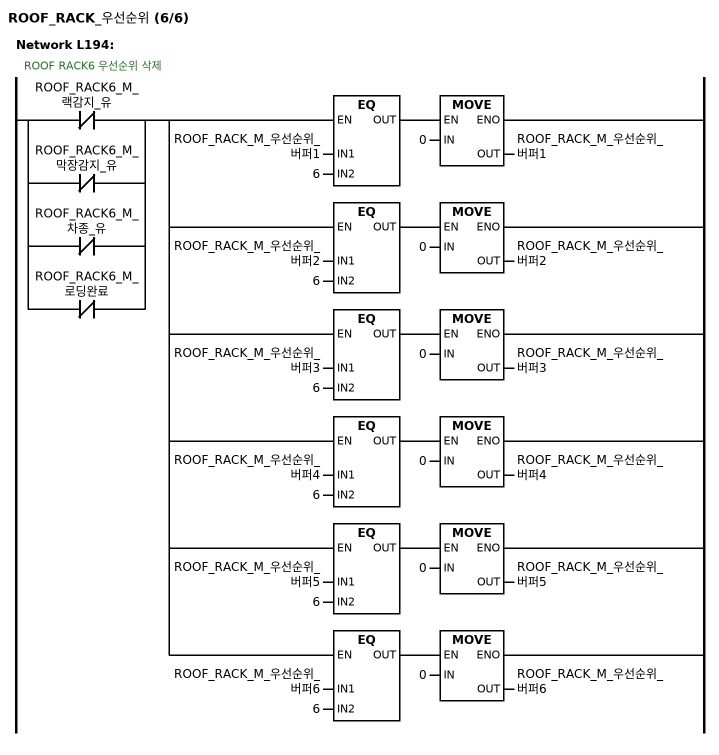
(* ROOF RACK6 우선순위 삭제 *)
(* Rung L194 *)
_p36 := NOT ROOF_RACK6_M_랙감지_유 OR NOT ROOF_RACK6_M_막장감지_유 OR NOT ROOF_RACK6_M_차종_유 OR NOT ROOF_RACK6_M_로딩완료;
IF _p36 THEN _t37 := ROOF_RACK_M_우선순위_버퍼1 = 6; END_IF;
IF _t37 THEN ROOF_RACK_M_우선순위_버퍼1 := 0; END_IF;
IF _p36 THEN _t38 := ROOF_RACK_M_우선순위_버퍼2 = 6; END_IF;
IF _t38 THEN ROOF_RACK_M_우선순위_버퍼2 := 0; END_IF;
IF _p36 THEN _t39 := ROOF_RACK_M_우선순위_버퍼3 = 6; END_IF;
IF _t39 THEN ROOF_RACK_M_우선순위_버퍼3 := 0; END_IF;
IF _p36 THEN _t40 := ROOF_RACK_M_우선순위_버퍼4 = 6; END_IF;
IF _t40 THEN ROOF_RACK_M_우선순위_버퍼4 := 0; END_IF;
IF _p36 THEN _t41 := ROOF_RACK_M_우선순위_버퍼5 = 6; END_IF;
IF _t41 THEN ROOF_RACK_M_우선순위_버퍼5 := 0; END_IF;
IF _p36 THEN _t42 := ROOF_RACK_M_우선순위_버퍼6 = 6; END_IF;
IF _t42 THEN ROOF_RACK_M_우선순위_버퍼6 := 0; END_IF;
END_PROGRAM

PROGRAM ROOF_RACK_차종비교 (* task: 스캔 프로그램 *)
VAR_EXTERNAL RETAIN
    R361_1_M_RACK3_동일차종 : BOOL; (* AT %MW1565.2 *)
    R361_1_M_RACK4_동일차종 : BOOL; (* AT %MW1565.3 *)
    R361_1_M_RACK5_동일차종 : BOOL; (* AT %MW1565.4 *)
    R361_1_M_RACK6_동일차종 : BOOL; (* AT %MW1565.5 *)
    R361_1_M_기동_랙번호 : WORD; (* AT %MW1534 *)
    R361_1_M_부품비교차종 : WORD; (* AT %MW1532 *)
    R361_1_M_차종6_썬루프 : BOOL; (* AT %MW10003.4 *) (* R361 1 M 차종6 썬루프 *)
    R361_1_M_차종6_일반루프 : BOOL; (* AT %MW10003.3 *) (* R361 1 M 차종6 일반루프 *)
    R361_1_M_차종_OPT1_R_RACK_무 : BOOL; (* AT %MW10005.3 *) (* R361 1 M 차종 OPT1 R RACK 무 *)
    R361_1_M_차종_유 : BOOL; (* AT %MW1502.0 *)
    R361_2_M_RACK1_동일차종 : BOOL; (* AT %MW1565.0 *)
    R361_2_M_RACK2_동일차종 : BOOL; (* AT %MW1565.1 *)
    R361_2_M_기동_랙번호 : WORD; (* AT %MW1535 *)
    R361_2_M_부품비교차종 : WORD; (* AT %MW1533 *)
    R361_2_M_차종6_썬루프 : BOOL; (* AT %MW10023.4 *) (* R361 2 M 차종6 썬루프 *)
    R361_2_M_차종6_일반루프 : BOOL; (* AT %MW10023.3 *) (* R361 2 M 차종6 일반루프 *)
    R361_2_M_차종_OPT1_R_RACK_유 : BOOL; (* AT %MW10025.2 *) (* R361 2 M 차종 OPT1 R RACK 유 *)
    R361_2_M_차종_유 : BOOL; (* AT %MW1502.2 *)
    ROOF_RACK1_M_우선순위_지정 : BOOL; (* AT %MW1564.0 *)
    ROOF_RACK1_M_차종 : WORD; (* AT %MW1541 *)
    ROOF_RACK2_M_우선순위_지정 : BOOL; (* AT %MW1564.1 *)
    ROOF_RACK2_M_차종 : WORD; (* AT %MW1542 *)
    ROOF_RACK3_M_우선순위_지정 : BOOL; (* AT %MW1564.2 *)
    ROOF_RACK3_M_차종 : WORD; (* AT %MW1543 *)
    ROOF_RACK4_M_우선순위_지정 : BOOL; (* AT %MW1564.3 *)
    ROOF_RACK4_M_차종 : WORD; (* AT %MW1544 *)
    ROOF_RACK5_M_우선순위_지정 : BOOL; (* AT %MW1564.4 *)
    ROOF_RACK5_M_차종 : WORD; (* AT %MW1545 *)
    ROOF_RACK6_M_우선순위_지정 : BOOL; (* AT %MW1564.5 *)
    ROOF_RACK6_M_차종 : WORD; (* AT %MW1546 *)
    ROOF_RACK_M_버퍼1_지정 : BOOL; (* AT %MW1562.0 *)
    ROOF_RACK_M_버퍼2_지정 : BOOL; (* AT %MW1562.1 *)
    ROOF_RACK_M_버퍼3_지정 : BOOL; (* AT %MW1562.2 *)
    ROOF_RACK_M_버퍼4_지정 : BOOL; (* AT %MW1562.3 *)
    ROOF_RACK_M_버퍼5_지정 : BOOL; (* AT %MW1562.4 *)
    ROOF_RACK_M_버퍼6_지정 : BOOL; (* AT %MW1562.5 *)
    ROOF_RACK_M_우선순위_버퍼1 : WORD; (* AT %MW1551 *)
    ROOF_RACK_M_우선순위_버퍼2 : WORD; (* AT %MW1552 *)
    ROOF_RACK_M_우선순위_버퍼3 : WORD; (* AT %MW1553 *)
    ROOF_RACK_M_우선순위_버퍼4 : WORD; (* AT %MW1554 *)
    ROOF_RACK_M_우선순위_버퍼5 : WORD; (* AT %MW1555 *)
    ROOF_RACK_M_우선순위_버퍼6 : WORD; (* AT %MW1556 *)
END_VAR
VAR
    _t1 : BOOL;
    _t2 : BOOL;
    _t3 : BOOL;
    _t4 : BOOL;
    _t5 : BOOL;
    _t6 : BOOL;
    _t7 : BOOL;
    _t8 : BOOL;
    _t9 : BOOL;
    _t10 : BOOL;
    _t11 : BOOL;
    _t12 : BOOL;
    _t13 : BOOL;
    _t14 : BOOL;
    _t15 : BOOL;
    _t16 : BOOL;
    _t17 : BOOL;
    _t18 : BOOL;
    _t19 : BOOL;
    _t20 : BOOL;
    _t21 : BOOL;
    _t22 : BOOL;
    _t23 : BOOL;
    _t24 : BOOL;
    _t25 : BOOL;
    _t26 : BOOL;
    _p27 : BOOL;
    _t28 : BOOL;
    _t29 : BOOL;
    _t30 : BOOL;
    _t31 : BOOL;
    _t32 : BOOL;
    _t33 : BOOL;
    _t34 : BOOL;
    _t35 : BOOL;
    _t36 : BOOL;
    _t37 : BOOL;
    _t38 : BOOL;
    _t39 : BOOL;
    _t40 : BOOL;
    _t41 : BOOL;
    _p42 : BOOL;
    _t43 : BOOL;
    _t44 : BOOL;
    _t45 : BOOL;
    _t46 : BOOL;
    _t47 : BOOL;
    _t48 : BOOL;
    _t49 : BOOL;
    _t50 : BOOL;
    _t51 : BOOL;
    _t52 : BOOL;
    _t53 : BOOL;
    _t54 : BOOL;
    _t55 : BOOL;
    _t56 : BOOL;
    _p57 : BOOL;
    _t58 : BOOL;
    _t59 : BOOL;
    _t60 : BOOL;
    _t61 : BOOL;
    _t62 : BOOL;
    _t63 : BOOL;
    _t64 : BOOL;
    _t65 : BOOL;
    _t66 : BOOL;
    _t67 : BOOL;
    _t68 : BOOL;
    _t69 : BOOL;
    _t70 : BOOL;
    _t71 : BOOL;
    _p72 : BOOL;
    _t73 : BOOL;
    _t74 : BOOL;
    _t75 : BOOL;
    _t76 : BOOL;
    _t77 : BOOL;
    _t78 : BOOL;
    _t79 : BOOL;
    _t80 : BOOL;
    _t81 : BOOL;
    _t82 : BOOL;
    _t83 : BOOL;
    _t84 : BOOL;
    _t85 : BOOL;
    _t86 : BOOL;
    _t87 : BOOL;
    _t88 : BOOL;
    _t89 : BOOL;
    _t90 : BOOL;
    _t91 : BOOL;
    _t92 : BOOL;
    _t93 : BOOL;
    _t94 : BOOL;
    _t95 : BOOL;
    _t96 : BOOL;
    _t97 : BOOL;
    _t98 : BOOL;
END_VAR

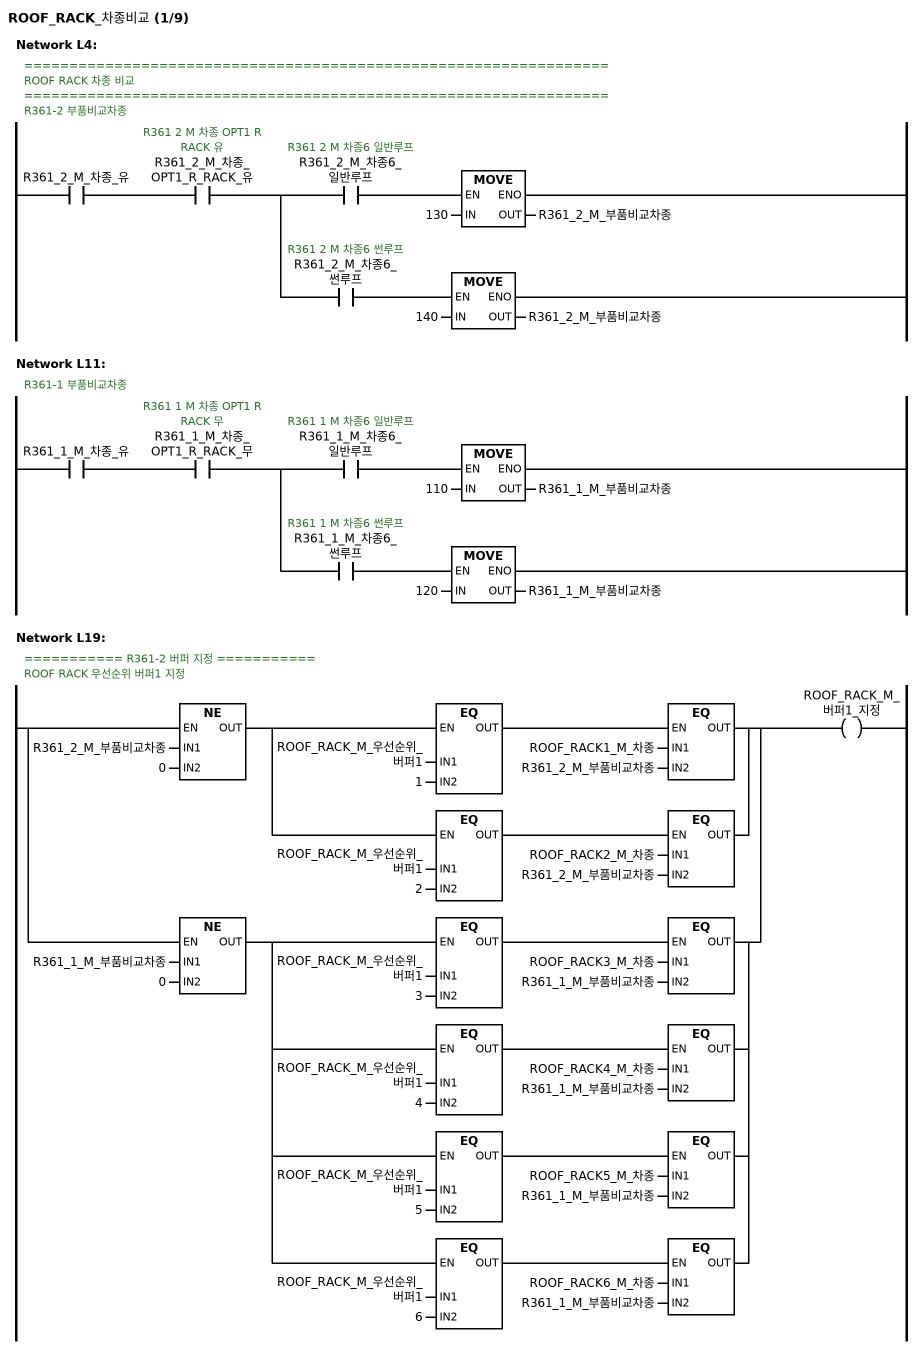
(* ================================================================= *)
(* ROOF RACK 차종 비교 *)
(* ================================================================= *)
(* R361-2 부품비교차종 *)
(* Rung L4 *)
IF R361_2_M_차종_유 AND R361_2_M_차종_OPT1_R_RACK_유 AND R361_2_M_차종6_일반루프 THEN R361_2_M_부품비교차종 := 130; END_IF;
IF R361_2_M_차종_유 AND R361_2_M_차종_OPT1_R_RACK_유 AND R361_2_M_차종6_썬루프 THEN R361_2_M_부품비교차종 := 140; END_IF;
(* R361-1 부품비교차종 *)
(* Rung L11 *)
IF R361_1_M_차종_유 AND R361_1_M_차종_OPT1_R_RACK_무 AND R361_1_M_차종6_일반루프 THEN R361_1_M_부품비교차종 := 110; END_IF;
IF R361_1_M_차종_유 AND R361_1_M_차종_OPT1_R_RACK_무 AND R361_1_M_차종6_썬루프 THEN R361_1_M_부품비교차종 := 120; END_IF;
(* =========== R361-2 버퍼 지정 =========== *)
(* ROOF RACK 우선순위 버퍼1 지정 *)
(* Rung L19 *)
IF R361_2_M_부품비교차종 <> 0 THEN _t1 := ROOF_RACK_M_우선순위_버퍼1 = 1; END_IF;
IF _t1 THEN _t2 := ROOF_RACK1_M_차종 = R361_2_M_부품비교차종; END_IF;
IF R361_2_M_부품비교차종 <> 0 THEN _t3 := ROOF_RACK_M_우선순위_버퍼1 = 2; END_IF;
IF _t3 THEN _t4 := ROOF_RACK2_M_차종 = R361_2_M_부품비교차종; END_IF;
IF R361_1_M_부품비교차종 <> 0 THEN _t5 := ROOF_RACK_M_우선순위_버퍼1 = 3; END_IF;
IF _t5 THEN _t6 := ROOF_RACK3_M_차종 = R361_1_M_부품비교차종; END_IF;
IF R361_1_M_부품비교차종 <> 0 THEN _t7 := ROOF_RACK_M_우선순위_버퍼1 = 4; END_IF;
IF _t7 THEN _t8 := ROOF_RACK4_M_차종 = R361_1_M_부품비교차종; END_IF;
IF R361_1_M_부품비교차종 <> 0 THEN _t9 := ROOF_RACK_M_우선순위_버퍼1 = 5; END_IF;
IF _t9 THEN _t10 := ROOF_RACK5_M_차종 = R361_1_M_부품비교차종; END_IF;
IF R361_1_M_부품비교차종 <> 0 THEN _t11 := ROOF_RACK_M_우선순위_버퍼1 = 6; END_IF;
IF _t11 THEN _t12 := ROOF_RACK6_M_차종 = R361_1_M_부품비교차종; END_IF;
ROOF_RACK_M_버퍼1_지정 := _t2 OR _t4 OR _t6 OR _t8 OR _t10 OR _t12;

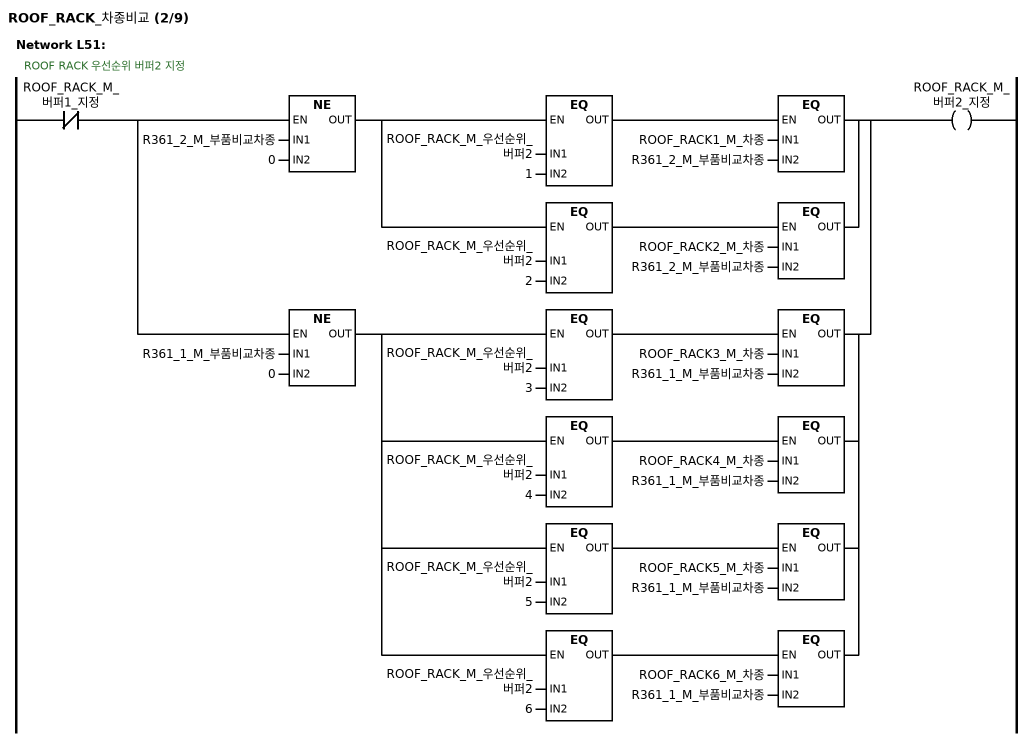
(* ROOF RACK 우선순위 버퍼2 지정 *)
(* Rung L51 *)
IF NOT ROOF_RACK_M_버퍼1_지정 THEN _t13 := R361_2_M_부품비교차종 <> 0; END_IF;
IF _t13 THEN _t14 := ROOF_RACK_M_우선순위_버퍼2 = 1; END_IF;
IF _t14 THEN _t15 := ROOF_RACK1_M_차종 = R361_2_M_부품비교차종; END_IF;
IF _t13 THEN _t16 := ROOF_RACK_M_우선순위_버퍼2 = 2; END_IF;
IF _t16 THEN _t17 := ROOF_RACK2_M_차종 = R361_2_M_부품비교차종; END_IF;
IF NOT ROOF_RACK_M_버퍼1_지정 THEN _t18 := R361_1_M_부품비교차종 <> 0; END_IF;
IF _t18 THEN _t19 := ROOF_RACK_M_우선순위_버퍼2 = 3; END_IF;
IF _t19 THEN _t20 := ROOF_RACK3_M_차종 = R361_1_M_부품비교차종; END_IF;
IF _t18 THEN _t21 := ROOF_RACK_M_우선순위_버퍼2 = 4; END_IF;
IF _t21 THEN _t22 := ROOF_RACK4_M_차종 = R361_1_M_부품비교차종; END_IF;
IF _t18 THEN _t23 := ROOF_RACK_M_우선순위_버퍼2 = 5; END_IF;
IF _t23 THEN _t24 := ROOF_RACK5_M_차종 = R361_1_M_부품비교차종; END_IF;
IF _t18 THEN _t25 := ROOF_RACK_M_우선순위_버퍼2 = 6; END_IF;
IF _t25 THEN _t26 := ROOF_RACK6_M_차종 = R361_1_M_부품비교차종; END_IF;
ROOF_RACK_M_버퍼2_지정 := _t15 OR _t17 OR _t20 OR _t22 OR _t24 OR _t26;

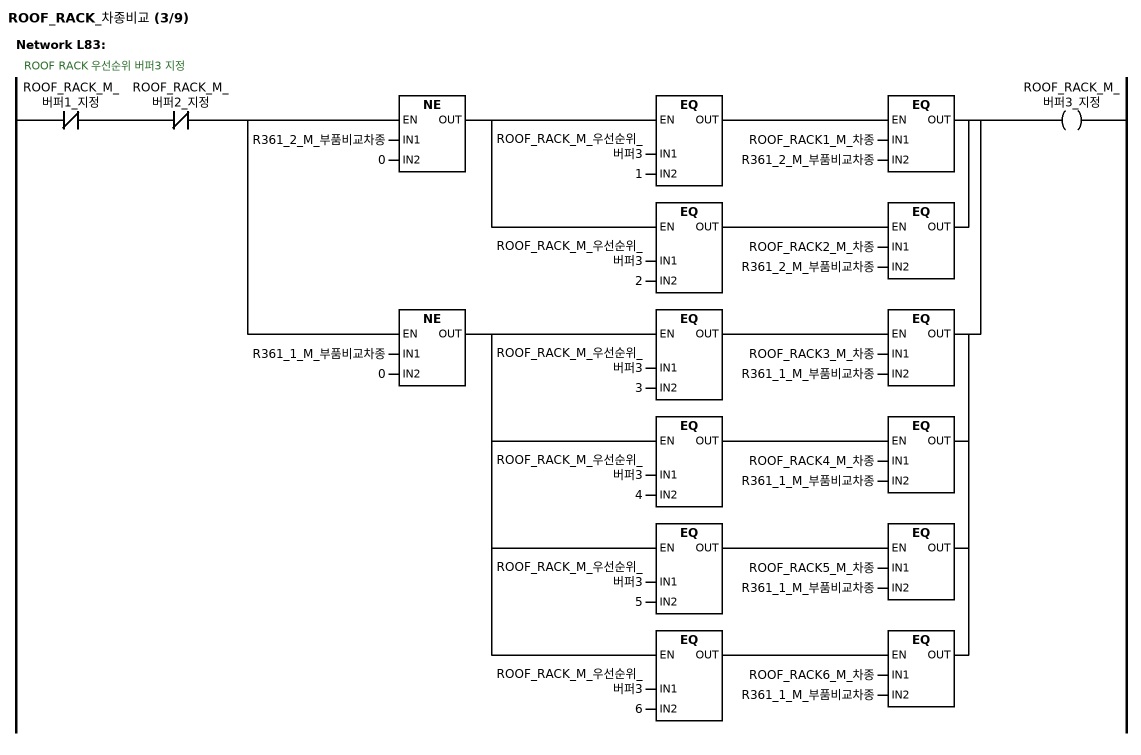
(* ROOF RACK 우선순위 버퍼3 지정 *)
(* Rung L83 *)
_p27 := NOT ROOF_RACK_M_버퍼1_지정 AND NOT ROOF_RACK_M_버퍼2_지정;
IF _p27 THEN _t28 := R361_2_M_부품비교차종 <> 0; END_IF;
IF _t28 THEN _t29 := ROOF_RACK_M_우선순위_버퍼3 = 1; END_IF;
IF _t29 THEN _t30 := ROOF_RACK1_M_차종 = R361_2_M_부품비교차종; END_IF;
IF _t28 THEN _t31 := ROOF_RACK_M_우선순위_버퍼3 = 2; END_IF;
IF _t31 THEN _t32 := ROOF_RACK2_M_차종 = R361_2_M_부품비교차종; END_IF;
IF _p27 THEN _t33 := R361_1_M_부품비교차종 <> 0; END_IF;
IF _t33 THEN _t34 := ROOF_RACK_M_우선순위_버퍼3 = 3; END_IF;
IF _t34 THEN _t35 := ROOF_RACK3_M_차종 = R361_1_M_부품비교차종; END_IF;
IF _t33 THEN _t36 := ROOF_RACK_M_우선순위_버퍼3 = 4; END_IF;
IF _t36 THEN _t37 := ROOF_RACK4_M_차종 = R361_1_M_부품비교차종; END_IF;
IF _t33 THEN _t38 := ROOF_RACK_M_우선순위_버퍼3 = 5; END_IF;
IF _t38 THEN _t39 := ROOF_RACK5_M_차종 = R361_1_M_부품비교차종; END_IF;
IF _t33 THEN _t40 := ROOF_RACK_M_우선순위_버퍼3 = 6; END_IF;
IF _t40 THEN _t41 := ROOF_RACK6_M_차종 = R361_1_M_부품비교차종; END_IF;
ROOF_RACK_M_버퍼3_지정 := _t30 OR _t32 OR _t35 OR _t37 OR _t39 OR _t41;

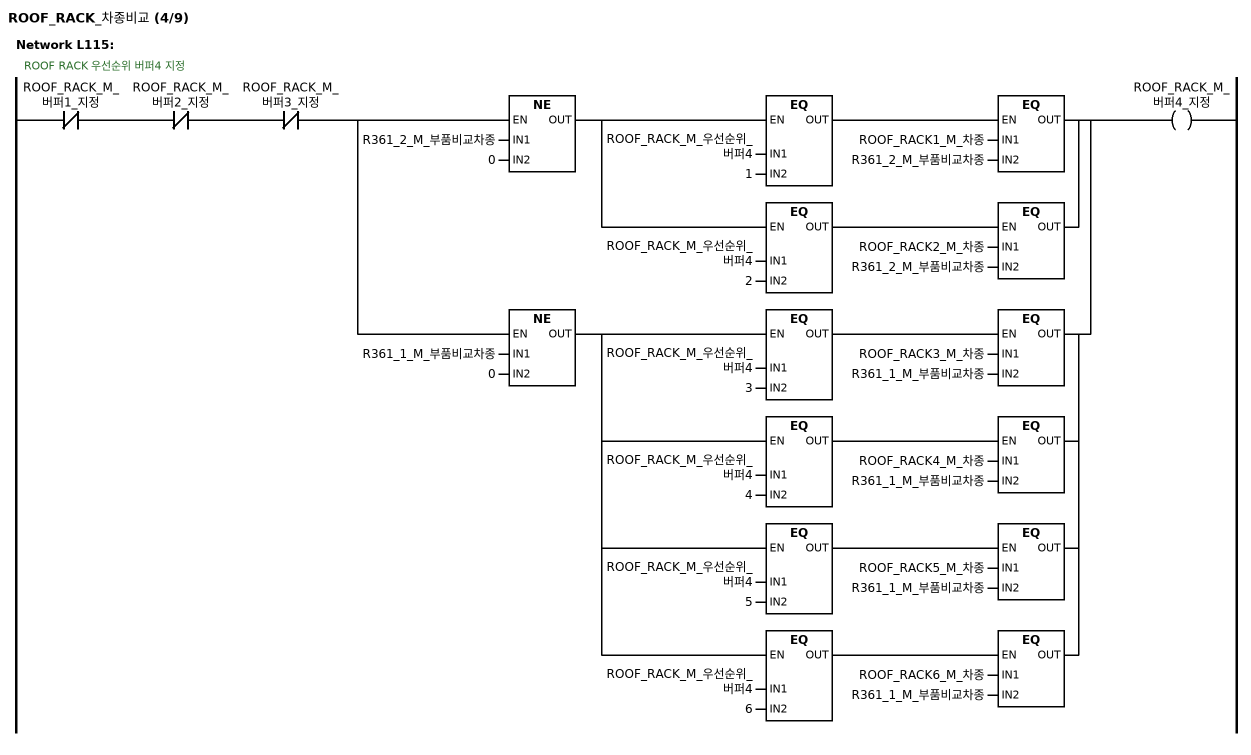
(* ROOF RACK 우선순위 버퍼4 지정 *)
(* Rung L115 *)
_p42 := NOT ROOF_RACK_M_버퍼1_지정 AND NOT ROOF_RACK_M_버퍼2_지정 AND NOT ROOF_RACK_M_버퍼3_지정;
IF _p42 THEN _t43 := R361_2_M_부품비교차종 <> 0; END_IF;
IF _t43 THEN _t44 := ROOF_RACK_M_우선순위_버퍼4 = 1; END_IF;
IF _t44 THEN _t45 := ROOF_RACK1_M_차종 = R361_2_M_부품비교차종; END_IF;
IF _t43 THEN _t46 := ROOF_RACK_M_우선순위_버퍼4 = 2; END_IF;
IF _t46 THEN _t47 := ROOF_RACK2_M_차종 = R361_2_M_부품비교차종; END_IF;
IF _p42 THEN _t48 := R361_1_M_부품비교차종 <> 0; END_IF;
IF _t48 THEN _t49 := ROOF_RACK_M_우선순위_버퍼4 = 3; END_IF;
IF _t49 THEN _t50 := ROOF_RACK3_M_차종 = R361_1_M_부품비교차종; END_IF;
IF _t48 THEN _t51 := ROOF_RACK_M_우선순위_버퍼4 = 4; END_IF;
IF _t51 THEN _t52 := ROOF_RACK4_M_차종 = R361_1_M_부품비교차종; END_IF;
IF _t48 THEN _t53 := ROOF_RACK_M_우선순위_버퍼4 = 5; END_IF;
IF _t53 THEN _t54 := ROOF_RACK5_M_차종 = R361_1_M_부품비교차종; END_IF;
IF _t48 THEN _t55 := ROOF_RACK_M_우선순위_버퍼4 = 6; END_IF;
IF _t55 THEN _t56 := ROOF_RACK6_M_차종 = R361_1_M_부품비교차종; END_IF;
ROOF_RACK_M_버퍼4_지정 := _t45 OR _t47 OR _t50 OR _t52 OR _t54 OR _t56;

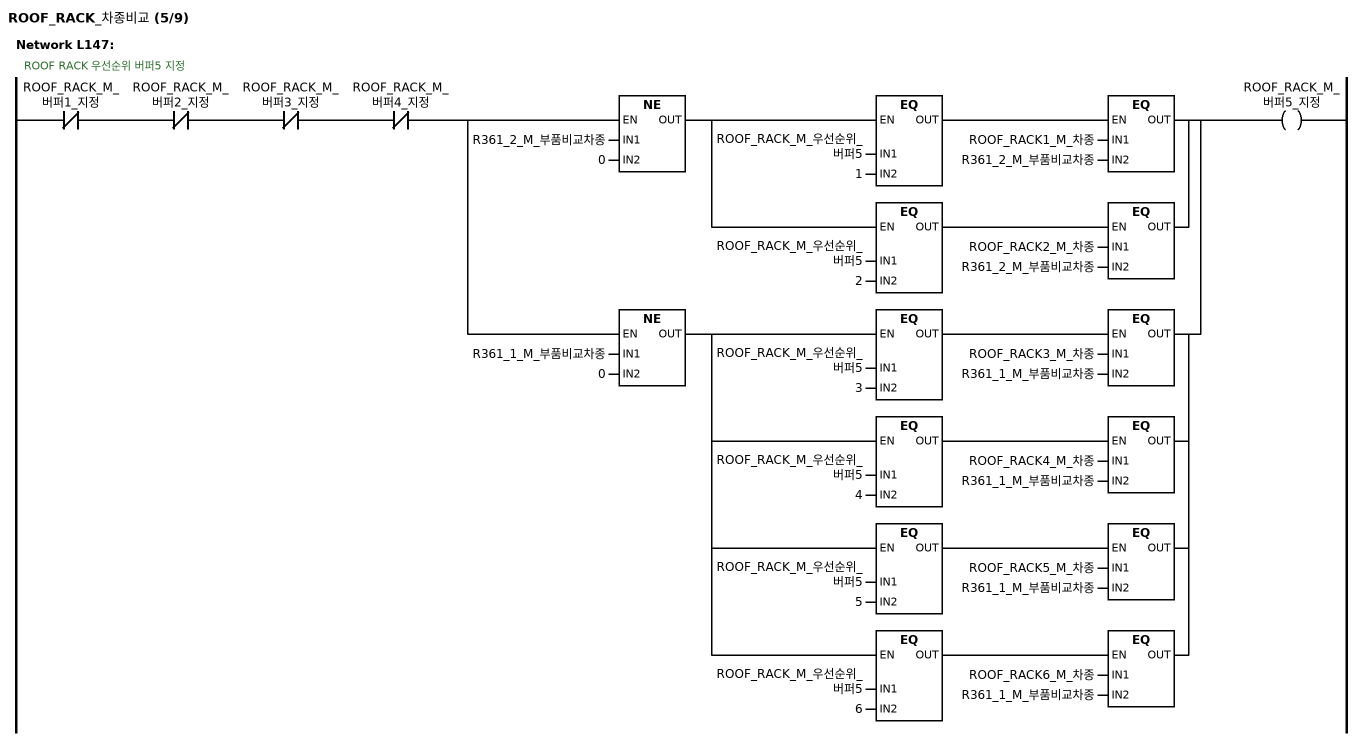
(* ROOF RACK 우선순위 버퍼5 지정 *)
(* Rung L147 *)
_p57 := NOT ROOF_RACK_M_버퍼1_지정 AND NOT ROOF_RACK_M_버퍼2_지정 AND NOT ROOF_RACK_M_버퍼3_지정 AND NOT ROOF_RACK_M_버퍼4_지정;
IF _p57 THEN _t58 := R361_2_M_부품비교차종 <> 0; END_IF;
IF _t58 THEN _t59 := ROOF_RACK_M_우선순위_버퍼5 = 1; END_IF;
IF _t59 THEN _t60 := ROOF_RACK1_M_차종 = R361_2_M_부품비교차종; END_IF;
IF _t58 THEN _t61 := ROOF_RACK_M_우선순위_버퍼5 = 2; END_IF;
IF _t61 THEN _t62 := ROOF_RACK2_M_차종 = R361_2_M_부품비교차종; END_IF;
IF _p57 THEN _t63 := R361_1_M_부품비교차종 <> 0; END_IF;
IF _t63 THEN _t64 := ROOF_RACK_M_우선순위_버퍼5 = 3; END_IF;
IF _t64 THEN _t65 := ROOF_RACK3_M_차종 = R361_1_M_부품비교차종; END_IF;
IF _t63 THEN _t66 := ROOF_RACK_M_우선순위_버퍼5 = 4; END_IF;
IF _t66 THEN _t67 := ROOF_RACK4_M_차종 = R361_1_M_부품비교차종; END_IF;
IF _t63 THEN _t68 := ROOF_RACK_M_우선순위_버퍼5 = 5; END_IF;
IF _t68 THEN _t69 := ROOF_RACK5_M_차종 = R361_1_M_부품비교차종; END_IF;
IF _t63 THEN _t70 := ROOF_RACK_M_우선순위_버퍼5 = 6; END_IF;
IF _t70 THEN _t71 := ROOF_RACK6_M_차종 = R361_1_M_부품비교차종; END_IF;
ROOF_RACK_M_버퍼5_지정 := _t60 OR _t62 OR _t65 OR _t67 OR _t69 OR _t71;

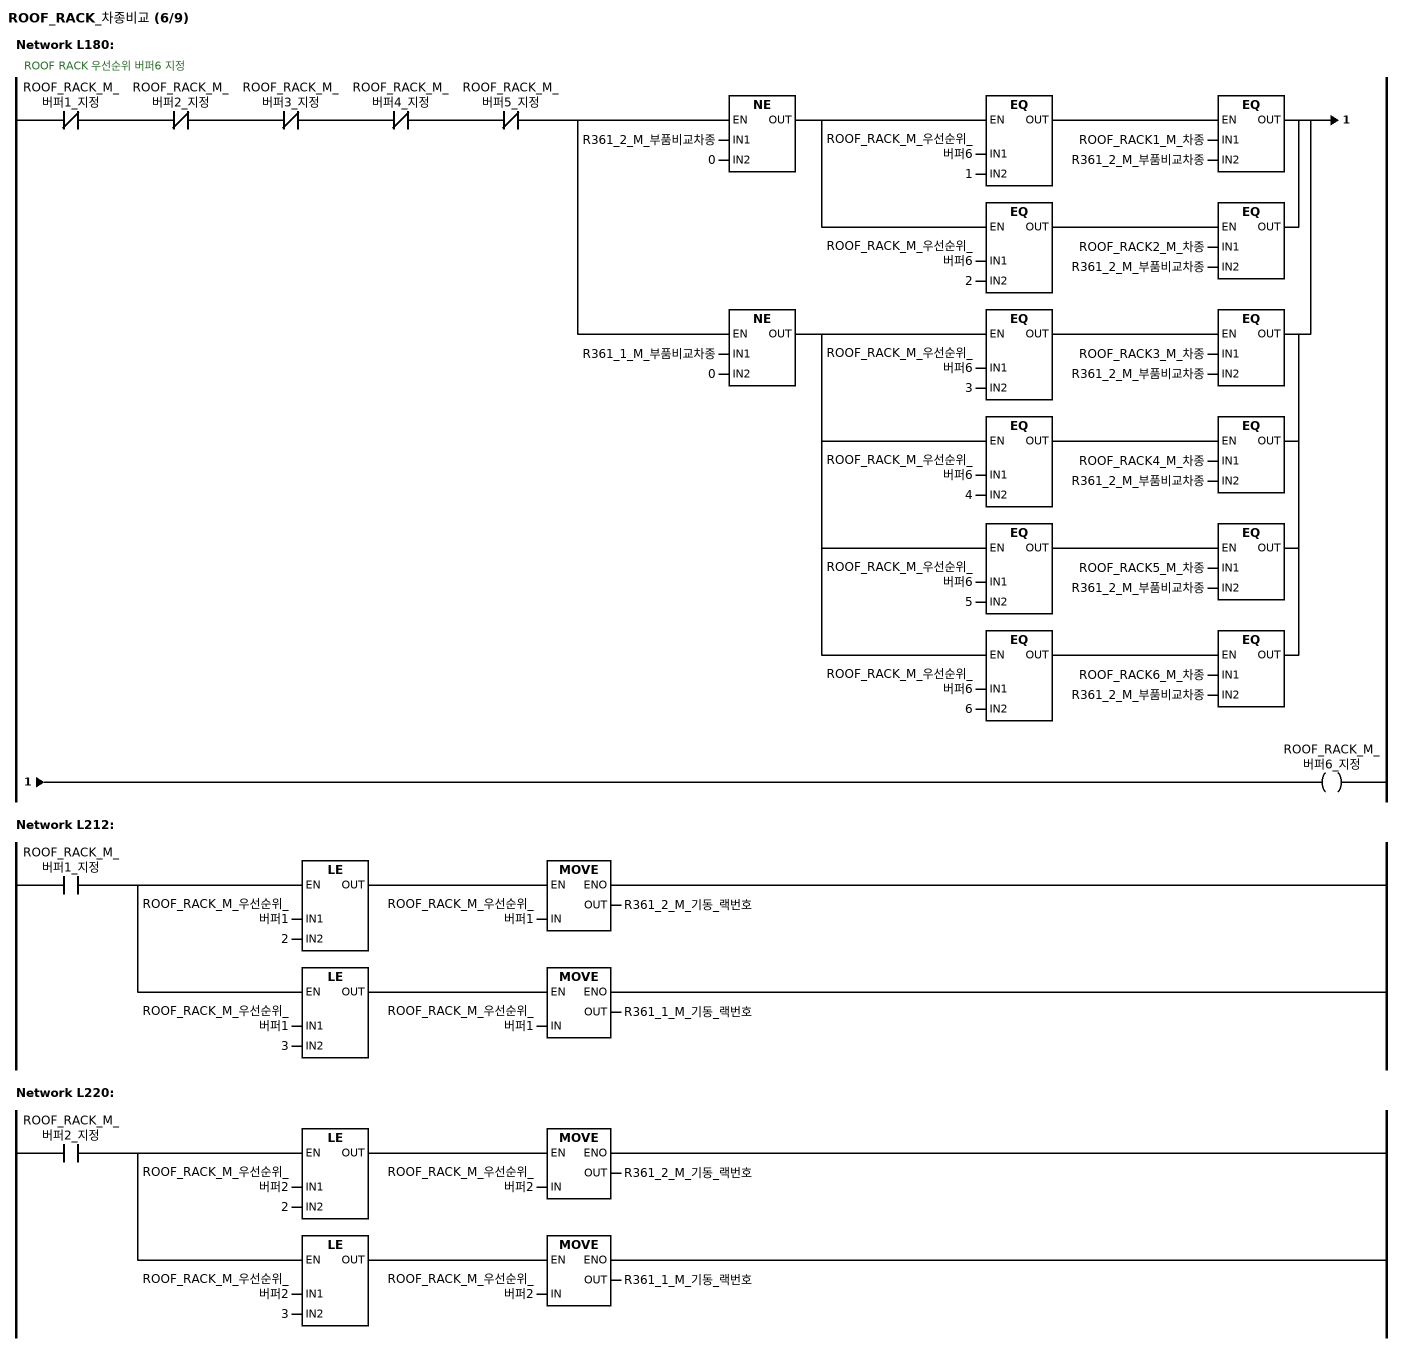
(* ROOF RACK 우선순위 버퍼6 지정 *)
(* Rung L180 *)
_p72 := NOT ROOF_RACK_M_버퍼1_지정 AND NOT ROOF_RACK_M_버퍼2_지정 AND NOT ROOF_RACK_M_버퍼3_지정 AND NOT ROOF_RACK_M_버퍼4_지정 AND NOT ROOF_RACK_M_버퍼5_지정;
IF _p72 THEN _t73 := R361_2_M_부품비교차종 <> 0; END_IF;
IF _t73 THEN _t74 := ROOF_RACK_M_우선순위_버퍼6 = 1; END_IF;
IF _t74 THEN _t75 := ROOF_RACK1_M_차종 = R361_2_M_부품비교차종; END_IF;
IF _t73 THEN _t76 := ROOF_RACK_M_우선순위_버퍼6 = 2; END_IF;
IF _t76 THEN _t77 := ROOF_RACK2_M_차종 = R361_2_M_부품비교차종; END_IF;
IF _p72 THEN _t78 := R361_1_M_부품비교차종 <> 0; END_IF;
IF _t78 THEN _t79 := ROOF_RACK_M_우선순위_버퍼6 = 3; END_IF;
IF _t79 THEN _t80 := ROOF_RACK3_M_차종 = R361_2_M_부품비교차종; END_IF;
IF _t78 THEN _t81 := ROOF_RACK_M_우선순위_버퍼6 = 4; END_IF;
IF _t81 THEN _t82 := ROOF_RACK4_M_차종 = R361_2_M_부품비교차종; END_IF;
IF _t78 THEN _t83 := ROOF_RACK_M_우선순위_버퍼6 = 5; END_IF;
IF _t83 THEN _t84 := ROOF_RACK5_M_차종 = R361_2_M_부품비교차종; END_IF;
IF _t78 THEN _t85 := ROOF_RACK_M_우선순위_버퍼6 = 6; END_IF;
IF _t85 THEN _t86 := ROOF_RACK6_M_차종 = R361_2_M_부품비교차종; END_IF;
ROOF_RACK_M_버퍼6_지정 := _t75 OR _t77 OR _t80 OR _t82 OR _t84 OR _t86;
(* Rung L212 *)
IF ROOF_RACK_M_버퍼1_지정 THEN _t87 := ROOF_RACK_M_우선순위_버퍼1 <= 2; END_IF;
IF _t87 THEN R361_2_M_기동_랙번호 := ROOF_RACK_M_우선순위_버퍼1; END_IF;
IF ROOF_RACK_M_버퍼1_지정 THEN _t88 := ROOF_RACK_M_우선순위_버퍼1 <= 3; END_IF;
IF _t88 THEN R361_1_M_기동_랙번호 := ROOF_RACK_M_우선순위_버퍼1; END_IF;
(* Rung L220 *)
IF ROOF_RACK_M_버퍼2_지정 THEN _t89 := ROOF_RACK_M_우선순위_버퍼2 <= 2; END_IF;
IF _t89 THEN R361_2_M_기동_랙번호 := ROOF_RACK_M_우선순위_버퍼2; END_IF;
IF ROOF_RACK_M_버퍼2_지정 THEN _t90 := ROOF_RACK_M_우선순위_버퍼2 <= 3; END_IF;
IF _t90 THEN R361_1_M_기동_랙번호 := ROOF_RACK_M_우선순위_버퍼2; END_IF;

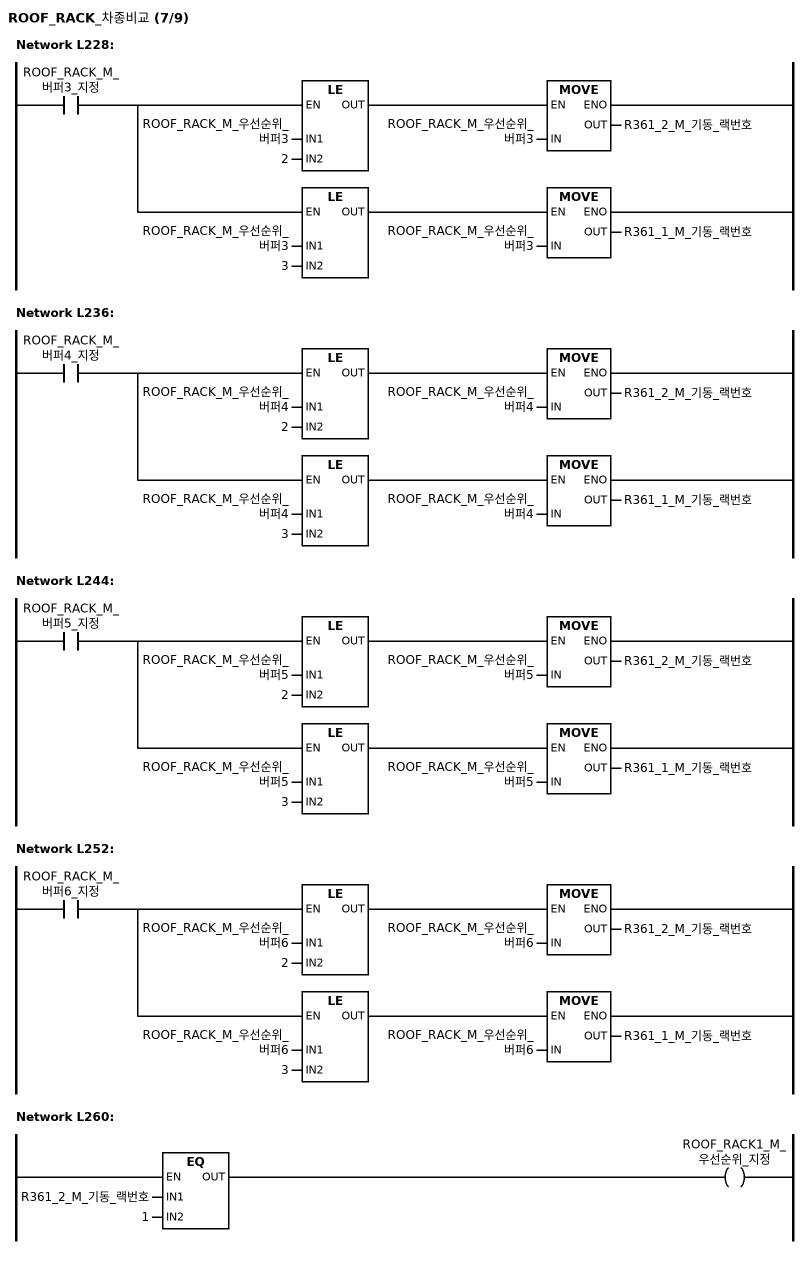
(* Rung L228 *)
IF ROOF_RACK_M_버퍼3_지정 THEN _t91 := ROOF_RACK_M_우선순위_버퍼3 <= 2; END_IF;
IF _t91 THEN R361_2_M_기동_랙번호 := ROOF_RACK_M_우선순위_버퍼3; END_IF;
IF ROOF_RACK_M_버퍼3_지정 THEN _t92 := ROOF_RACK_M_우선순위_버퍼3 <= 3; END_IF;
IF _t92 THEN R361_1_M_기동_랙번호 := ROOF_RACK_M_우선순위_버퍼3; END_IF;
(* Rung L236 *)
IF ROOF_RACK_M_버퍼4_지정 THEN _t93 := ROOF_RACK_M_우선순위_버퍼4 <= 2; END_IF;
IF _t93 THEN R361_2_M_기동_랙번호 := ROOF_RACK_M_우선순위_버퍼4; END_IF;
IF ROOF_RACK_M_버퍼4_지정 THEN _t94 := ROOF_RACK_M_우선순위_버퍼4 <= 3; END_IF;
IF _t94 THEN R361_1_M_기동_랙번호 := ROOF_RACK_M_우선순위_버퍼4; END_IF;
(* Rung L244 *)
IF ROOF_RACK_M_버퍼5_지정 THEN _t95 := ROOF_RACK_M_우선순위_버퍼5 <= 2; END_IF;
IF _t95 THEN R361_2_M_기동_랙번호 := ROOF_RACK_M_우선순위_버퍼5; END_IF;
IF ROOF_RACK_M_버퍼5_지정 THEN _t96 := ROOF_RACK_M_우선순위_버퍼5 <= 3; END_IF;
IF _t96 THEN R361_1_M_기동_랙번호 := ROOF_RACK_M_우선순위_버퍼5; END_IF;
(* Rung L252 *)
IF ROOF_RACK_M_버퍼6_지정 THEN _t97 := ROOF_RACK_M_우선순위_버퍼6 <= 2; END_IF;
IF _t97 THEN R361_2_M_기동_랙번호 := ROOF_RACK_M_우선순위_버퍼6; END_IF;
IF ROOF_RACK_M_버퍼6_지정 THEN _t98 := ROOF_RACK_M_우선순위_버퍼6 <= 3; END_IF;
IF _t98 THEN R361_1_M_기동_랙번호 := ROOF_RACK_M_우선순위_버퍼6; END_IF;
(* Rung L260 *)
ROOF_RACK1_M_우선순위_지정 := R361_2_M_기동_랙번호 = 1;

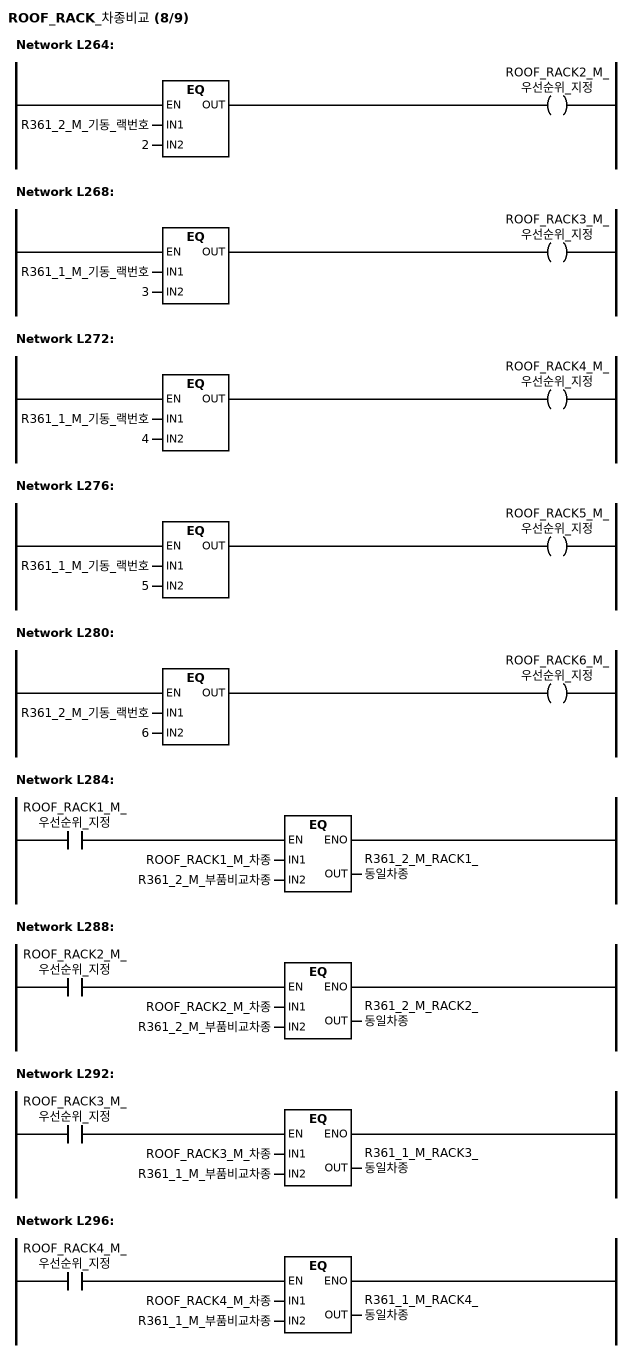
(* Rung L264 *)
ROOF_RACK2_M_우선순위_지정 := R361_2_M_기동_랙번호 = 2;
(* Rung L268 *)
ROOF_RACK3_M_우선순위_지정 := R361_1_M_기동_랙번호 = 3;
(* Rung L272 *)
ROOF_RACK4_M_우선순위_지정 := R361_1_M_기동_랙번호 = 4;
(* Rung L276 *)
ROOF_RACK5_M_우선순위_지정 := R361_1_M_기동_랙번호 = 5;
(* Rung L280 *)
ROOF_RACK6_M_우선순위_지정 := R361_2_M_기동_랙번호 = 6;
(* Rung L284 *)
IF ROOF_RACK1_M_우선순위_지정 THEN R361_2_M_RACK1_동일차종 := ROOF_RACK1_M_차종 = R361_2_M_부품비교차종; END_IF;
(* Rung L288 *)
IF ROOF_RACK2_M_우선순위_지정 THEN R361_2_M_RACK2_동일차종 := ROOF_RACK2_M_차종 = R361_2_M_부품비교차종; END_IF;
(* Rung L292 *)
IF ROOF_RACK3_M_우선순위_지정 THEN R361_1_M_RACK3_동일차종 := ROOF_RACK3_M_차종 = R361_1_M_부품비교차종; END_IF;
(* Rung L296 *)
IF ROOF_RACK4_M_우선순위_지정 THEN R361_1_M_RACK4_동일차종 := ROOF_RACK4_M_차종 = R361_1_M_부품비교차종; END_IF;

